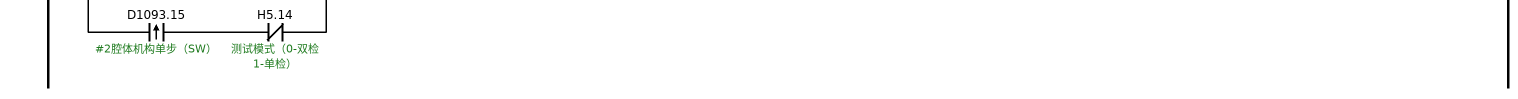
; [picture p240: 氦检机构 / 氦检腔2自动, rungs 7-7]
; rung 7: #2腔体机构步进条件（自动步）
LD D1096.00  ; #2腔体机构自动开始（自动步）
AND T1550  ; #2腔体机构开始运行条件延时(自动步)
LD D1096.01  ; #2腔体机构平移气缸到氦检位/数据初始化（自动步）
ANDNOT 802.01  ; #2腔体平移一级气缸缩回位标志[0002.01]
AND 802.02  ; #2腔体平移一级气缸伸出位标志[0002.02]
AND 802.03  ; #2腔体平移二级气缸缩回位标志[0002.03]
ANDNOT 802.04  ; #2腔体平移二级气缸伸出位标志[0002.04]
AND T1551  ; #2腔体机构数据初始化延时（自动步）
ORLD
LD D1096.02  ; #2腔体机构腔体顶升气缸上升（自动步）
AND 802.05  ; #2腔体顶伸气缸上升位标志[0002.05]
ANDNOT 802.06  ; #2腔体顶伸气缸下降位标志[0002.06]
ORLD
LD D1096.03  ; #2腔体机构等待氦检阀打开条件及腔体抽气阀打开条件/开腔体阀（自动步）
AND 821.10  ; #2-1腔体阀开到位标志
AND 821.12  ; #2-2腔体阀开到位标志
ANDNOT H27.00  ; #1腔体有清氦需求
ANDNOT H37.00  ; #3腔体有清氦需求
AND D1092.15  ; #2腔体机构腔体抽气阀打开允许
AND D1092.14  ; #2腔体氦检阀打开允许条件
LD W380.15  ; 氦检仪漏率低于设定值（稳态）
OR H5.02  ; 氦检仪屏蔽
ANDLD
AND=L(301) D1104 #0  ; #2腔体机构清氦步序号
ORLD
OR D1096.04  ; #2腔体机构（自动步）
LD D1096.05  ; #2腔体机构腔体抽气阀打开/延时开电池抽气阀（自动步）
LD T2000  ; #2-1腔体抽真空阈值到达延时（测试）
LD 823.08  ; #2-1电池抽真空阀开到位标志
AND T2020  ; #2-1电池抽真空阈值到达延时（测试）
LD H31.00  ; #2-1电池泄漏
ANDNOT H31.01  ; #2-2电池泄漏
ORLD
ORNOT H30.00  ; #2-1腔体有料记忆
LD 823.10  ; #2-2电池抽真空阀开到位标志
AND T2320  ; #2-2电池抽真空阈值到达延时（测试）
LDNOT H31.00  ; #2-1电池泄漏
AND H31.01  ; #2-2电池泄漏
ORLD
ORNOT H30.01  ; #2-2腔体有料记忆
ANDLD
OR H5.15  ; 腔体模式（0-正压 1-负压）
OR H5.10  ; 空跑程序
ANDLD
LD H31.04  ; #2-1腔体抽真空NG
ORNOT H30.00  ; #2-1腔体有料记忆
LD H31.05  ; #2-2腔体抽真空NG
ORNOT H30.01  ; #2-2腔体有料记忆
ANDLD
ORLD
LD H31.00  ; #2-1电池泄漏
AND H31.01  ; #2-2电池泄漏
ORLD
ANDLD
ORLD
LD D1096.06  ; #2腔体机构关电池抽气阀（自动步）  // 单个电池出现电池泄漏时，需将对应的腔体阀门关闭
ANDNOT W407.14  ; 设备氦气压力信号[alm]
ANDNOT W407.15  ; 精密调压阀信号[alm]
AND 823.09  ; #2-1电池抽真空阀关到位标志
AND 823.11  ; #2-2电池抽真空阀关到位标志
ANDNOT H31.04  ; #2-1腔体抽真空NG
ANDNOT H31.05  ; #2-2腔体抽真空NG
LD H31.00  ; #2-1电池泄漏
AND 821.11  ; #2-1腔体阀关到位标志
ORNOT H31.00  ; #2-1电池泄漏
ORNOT H30.00  ; #2-1腔体有料记忆
ANDLD
LD H31.01  ; #2-2电池泄漏
AND 821.13  ; #2-2腔体阀关到位标志
ORNOT H31.01  ; #2-2电池泄漏
ORNOT H30.01  ; #2-2腔体有料记忆
ANDLD
ORLD
LD D1096.07  ; #2腔体机构开电池注氦阀（自动步）  // 单个电池出现注氦超时时，需将对应的腔体阀门关闭
LD 823.12  ; #2-1电池注氦阀开到位标志
AND T2024  ; #2-1电池注氦压力到达延时（测试）
OR H31.00  ; #2-1电池泄漏
LD H31.02  ; #2-1电池注氦超时
AND 821.11  ; #2-1腔体阀关到位标志
ORLD
ORNOT H30.00  ; #2-1腔体有料记忆
LD 823.14  ; #2-2电池注氦阀开到位标志
AND T2324  ; #2-2电池注氦压力到达延时（测试）
OR H31.01  ; #2-2电池泄漏
LD H31.03  ; #2-2电池注氦超时
AND 821.13  ; #2-2腔体阀关到位标志
ORLD
ORNOT H30.01  ; #2-2腔体有料记忆
ANDLD
OR H5.15  ; 腔体模式（0-正压 1-负压）
OR H5.10  ; 空跑程序
ANDLD
ORLD
LD D1096.08  ; #2腔体机构关电池注氦阀（自动步）
AND 823.13  ; #2-1电池注氦阀关到位标志
AND 823.15  ; #2-2电池注氦阀关到位标志
LDNOT H31.03  ; #2-2电池注氦超时
ORNOT H31.02  ; #2-1电池注氦超时
ANDLD
ORLD
OR D1096.09  ; #2腔体机构（自动步）
LD D1096.10  ; #2腔体机构开腔体氦检阀/延时关腔体抽气阀（自动步）
LD T2006  ; #2-1腔体氦检数据取值判定延时（测试）
LD 820.10  ; 氦检仪真空阀开到位标志
AND 802.07  ; #2腔体氦检阀开到位标志[0002.07]
OR H5.02  ; 氦检仪屏蔽
ANDLD
LD H31.06  ; #2-1腔体氦检时腔体压力过高
AND H31.07  ; #2-2腔体氦检时腔体压力过高
ORLD
ANDLD
ORLD
OR D1096.11  ; #2腔体机构（自动步）
LD D1096.12  ; #2腔体机构关腔体氦检阀（自动步）
AND 802.08  ; #2腔体氦检阀关到位标志[0002.08]
ANDNOT 802.07  ; #2腔体氦检阀开到位标志[0002.07]
ORLD
OR D1096.13  ; #2腔体机构（自动步）
LD D1096.14  ; #2腔体机构开腔体#2-1腔体阀/开腔体#2-2腔体阀（自动步）
AND 821.10  ; #2-1腔体阀开到位标志
AND 821.12  ; #2-2腔体阀开到位标志
AND 802.08  ; #2腔体氦检阀关到位标志[0002.08]
ANDNOT H5.15  ; 腔体模式（0-正压 1-负压）
AND D1092.15  ; #2腔体机构腔体抽气阀打开允许
ORLD
LD D1096.15  ; #2腔体机构开腔体抽真空阀/开电池抽真空阀（自动步）
LD T2007  ; #2-1腔体抽残气压力到达延时（测试）
OR T2008  ; #2-1腔体抽残气时间上限到达延时（测试）
ANDLD
LD T2026  ; #2-1电池抽残气压力到达延时（测试）
OR T2027  ; #2-1电池抽残气时间上限到达延时（测试）
ORNOT H30.00  ; #2-1腔体有料记忆
LD T2326  ; #2-2电池抽残气压力到达延时（测试）
OR T2327  ; #2-2电池抽残气时间上限到达延时（测试）
ORNOT H30.01  ; #2-2腔体有料记忆
ANDLD
OR H5.10  ; 空跑程序
ANDLD
ORLD
LD D1097.00  ; #2腔体机构关腔体抽真空阀/关电池抽真空阀/开腔体阀（自动步）
AND 821.09  ; #2腔体抽真空阀关到位标志
AND 821.10  ; #2-1腔体阀开到位标志
AND 821.12  ; #2-2腔体阀开到位标志
AND 823.09  ; #2-1电池抽真空阀关到位标志
AND 823.11  ; #2-2电池抽真空阀关到位标志
ORLD
LD D1097.01  ; #2腔体机构清氦需求判定（自动步）
ANDNOT H32.00  ; #2腔体有清氦需求
ORLD
LD D1097.02  ; #2腔体机构开腔体破真空阀/开电池破真空阀（自动步）
AND T2002  ; #2-1腔体破真空阈值到达延时（测试）
LD T2022  ; #2-1电池破真空阈值到达延时（测试）
AND T2322  ; #2-2电池破真空阈值到达延时（测试）
OR H5.15  ; 腔体模式（0-正压 1-负压）
ANDLD
ORLD
LD D1097.03  ; #2腔体机构关腔体破真空阀/关电池破真空阀（自动步）
AND 821.15  ; #2腔体破真空阀关到位标志
AND 824.01  ; #2-1电池破真空阀关到位标志
AND 824.03  ; #2-2电池破真空阀关到位标志
ORLD
LD D1097.04  ; #2腔体机构复测需求判定（自动步）
ANDNOT H32.05  ; 腔体有复测需求
ORLD
OR D1097.05  ; #2腔体机构（自动步）
LD D1097.06  ; #2腔体机构腔体顶升气缸下降（自动步）
ANDNOT 802.05  ; #2腔体顶伸气缸上升位标志[0002.05]
AND 802.06  ; #2腔体顶伸气缸下降位标志[0002.06]
AND D1092.00  ; #2腔体机构平移气缸安全移动条件
LD H30.06  ; #2-1腔体测试完成记忆
ORNOT H30.00  ; #2-1腔体有料记忆
ANDLD
LD H30.07  ; #2-2腔体测试完成记忆
ORNOT H30.01  ; #2-2腔体有料记忆
ANDLD
ORLD
OR D1097.07  ; #2腔体机构（自动步）
LD D1097.08  ; #2腔体机构腔体平移气缸到出料位（自动步）
AND 802.01  ; #2腔体平移一级气缸缩回位标志[0002.01]
ANDNOT 802.02  ; #2腔体平移一级气缸伸出位标志[0002.02]
AND 802.03  ; #2腔体平移二级气缸缩回位标志[0002.03]
ANDNOT 802.04  ; #2腔体平移二级气缸伸出位标志[0002.04]
ORLD
LD D1097.09  ; #2腔体机构腔体等待取料完成信号（自动步）
ANDNOT H30.00  ; #2-1腔体有料记忆
ANDNOT H30.01  ; #2-2腔体有料记忆
AND D1092.00  ; #2腔体机构平移气缸安全移动条件
ORLD
OR D1097.10  ; #2腔体机构（自动步）
LD D1097.11  ; #2腔体机构平移气缸到上料位（自动步）
ANDNOT 802.01  ; #2腔体平移一级气缸缩回位标志[0002.01]
AND 802.02  ; #2腔体平移一级气缸伸出位标志[0002.02]
ANDNOT 802.03  ; #2腔体平移二级气缸缩回位标志[0002.03]
AND 802.04  ; #2腔体平移二级气缸伸出位标志[0002.04]
ORLD
OR D1097.12  ; #2腔体机构（自动步）
OR D1097.13  ; #2腔体机构（自动步）
OR D1097.14  ; #2腔体机构（自动步）
LD D1097.15  ; #2腔体机构循环结束（自动步）
AND P_Off
ORLD
LD D1094.01  ; #2腔体机构单步/自动循环运行中（自动步）
@LD D1093.15  ; #2腔体机构单步（SW）
ANDNOT H5.14  ; 测试模式（0-双检 1-单检）
ORLD
ANDLD
OUT D1095.01  ; #2腔体机构步进条件（自动步）

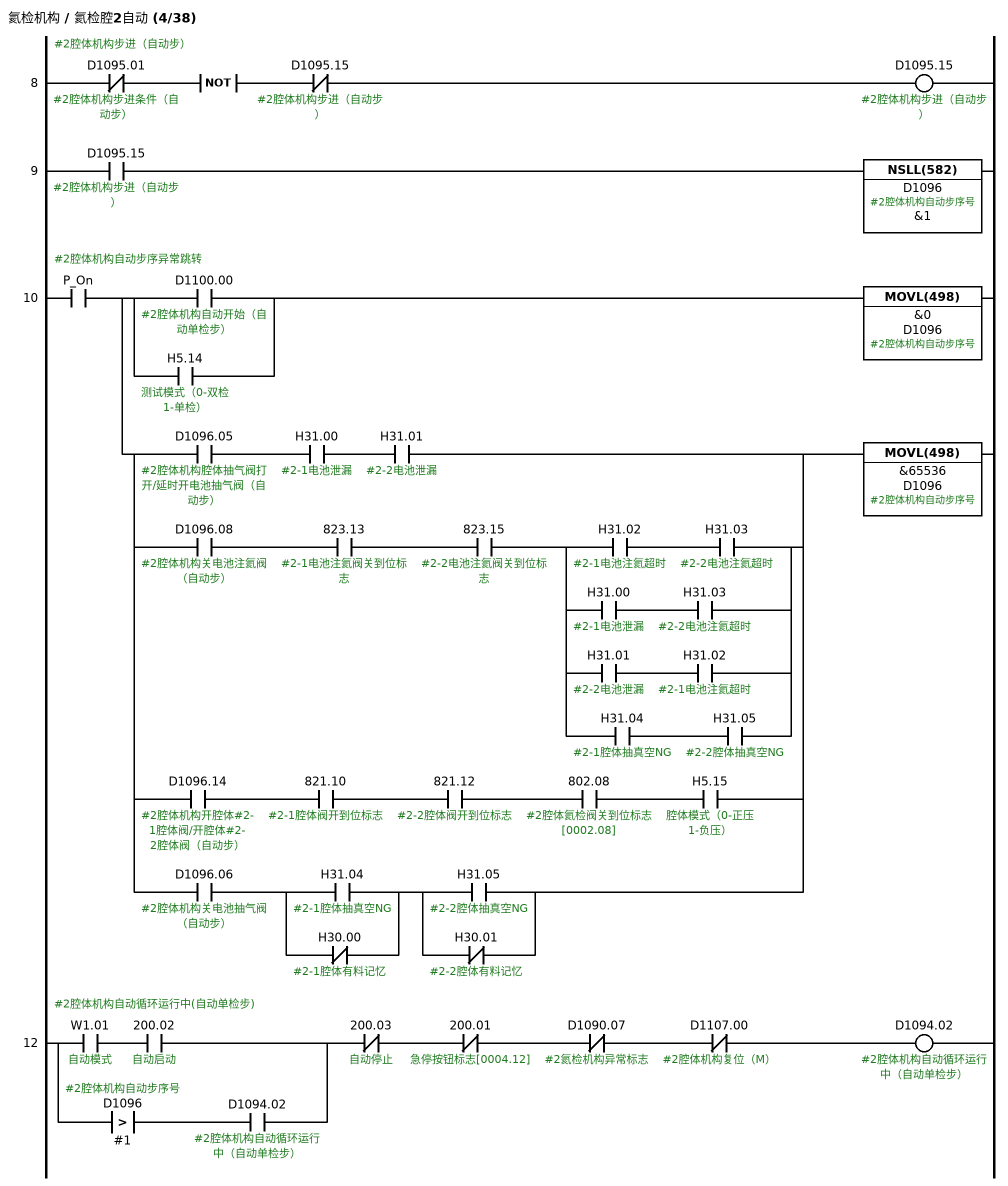
; rung 8: #2腔体机构步进（自动步）
LDNOT D1095.01  ; #2腔体机构步进条件（自动步）
NOT(520)
ANDNOT D1095.15  ; #2腔体机构步进（自动步）
OUT D1095.15  ; #2腔体机构步进（自动步）
; rung 9
LD D1095.15  ; #2腔体机构步进（自动步）
NSLL(582) D1096 &1  ; #2腔体机构自动步序号
; rung 10: #2腔体机构自动步序异常跳转
LD P_On
OUT TR0
LD D1100.00  ; #2腔体机构自动开始（自动单检步）
OR H5.14  ; 测试模式（0-双检 1-单检）
ANDLD
MOVL(498) &0 D1096  ; #2腔体机构自动步序号  // 测试模式为单检模式，腔体进入到复测步序时，将腔体机构自动步序清零
LD TR0
LD D1096.05  ; #2腔体机构腔体抽气阀打开/延时开电池抽气阀（自动步）
AND H31.00  ; #2-1电池泄漏
AND H31.01  ; #2-2电池泄漏
LD D1096.08  ; #2腔体机构关电池注氦阀（自动步）
AND 823.13  ; #2-1电池注氦阀关到位标志
AND 823.15  ; #2-2电池注氦阀关到位标志
LD H31.02  ; #2-1电池注氦超时
AND H31.03  ; #2-2电池注氦超时
LD H31.00  ; #2-1电池泄漏
AND H31.03  ; #2-2电池注氦超时
ORLD
LD H31.01  ; #2-2电池泄漏
AND H31.02  ; #2-1电池注氦超时
ORLD
LD H31.04  ; #2-1腔体抽真空NG
AND H31.05  ; #2-2腔体抽真空NG
ORLD
ANDLD
ORLD
LD D1096.14  ; #2腔体机构开腔体#2-1腔体阀/开腔体#2-2腔体阀（自动步）  // 负压模式不需要进行氦检后抽真空动作
AND 821.10  ; #2-1腔体阀开到位标志
AND 821.12  ; #2-2腔体阀开到位标志
AND 802.08  ; #2腔体氦检阀关到位标志[0002.08]
AND H5.15  ; 腔体模式（0-正压 1-负压）
ORLD
LD D1096.06  ; #2腔体机构关电池抽气阀（自动步）
LD H31.04  ; #2-1腔体抽真空NG
ORNOT H30.00  ; #2-1腔体有料记忆
ANDLD
LD H31.05  ; #2-2腔体抽真空NG
ORNOT H30.01  ; #2-2腔体有料记忆
ANDLD
ORLD
ANDLD
MOVL(498) &65536 D1096  ; #2腔体机构自动步序号  // 出现腔体抽真空NG，双电池抽真空NG，双电池注氦超时的情况，均跳转至自动步序D1067.0
; rung 11: ******************************* / 自动单检步序 / *******************************
; rung 12: #2腔体机构自动循环运行中(自动单检步)
LD W1.01  ; 自动模式
AND 200.02  ; 自动启动
LD>L(321) D1096 #1  ; #2腔体机构自动步序号
AND D1094.02  ; #2腔体机构自动循环运行中（自动单检步）
ORLD
ANDNOT 200.03  ; 自动停止
ANDNOT 200.01  ; 急停按钮标志[0004.12]
ANDNOT D1090.07  ; #2氦检机构异常标志
ANDNOT D1107.00  ; #2腔体机构复位（M）
OUT D1094.02  ; #2腔体机构自动循环运行中（自动单检步）

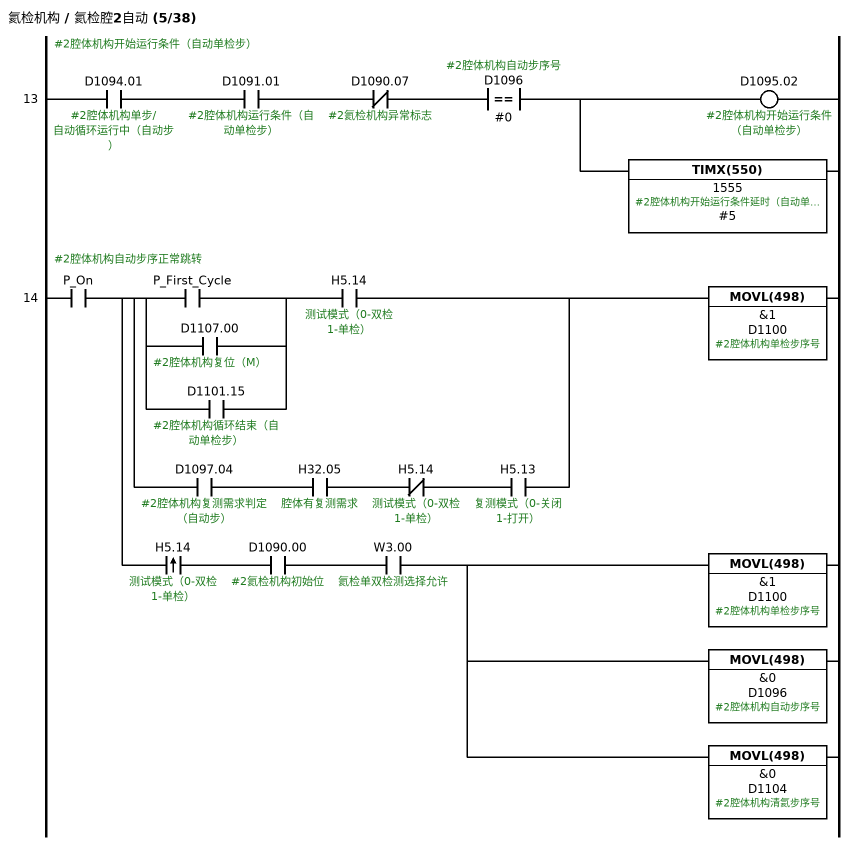
; rung 13: #2腔体机构开始运行条件（自动单检步）
LD D1094.01  ; #2腔体机构单步/自动循环运行中（自动步）
AND D1091.01  ; #2腔体机构运行条件（自动单检步）
ANDNOT D1090.07  ; #2氦检机构异常标志
AND=L(301) D1096 #0  ; #2腔体机构自动步序号
OUT D1095.02  ; #2腔体机构开始运行条件（自动单检步）
TIMX(550) 1555 #5  ; #2腔体机构开始运行条件延时（自动单检步）
; rung 14: #2腔体机构自动步序正常跳转
LD P_On
OUT TR0
LD P_First_Cycle
OR D1107.00  ; #2腔体机构复位（M）
OR D1101.15  ; #2腔体机构循环结束（自动单检步）
AND H5.14  ; 测试模式（0-双检 1-单检）
LD D1097.04  ; #2腔体机构复测需求判定（自动步）
AND H32.05  ; 腔体有复测需求
ANDNOT H5.14  ; 测试模式（0-双检 1-单检）
AND H5.13  ; 复测模式（0-关闭 1-打开）
ORLD
ANDLD
MOVL(498) &1 D1100  ; #2腔体机构单检步序号
LD TR0
@AND H5.14  ; 测试模式（0-双检 1-单检）
AND D1090.00  ; #2氦检机构初始位
AND W3.00  ; 氦检单双检测选择允许
MOVL(498) &1 D1100  ; #2腔体机构单检步序号
MOVL(498) &0 D1096  ; #2腔体机构自动步序号
MOVL(498) &0 D1104  ; #2腔体机构清氦步序号

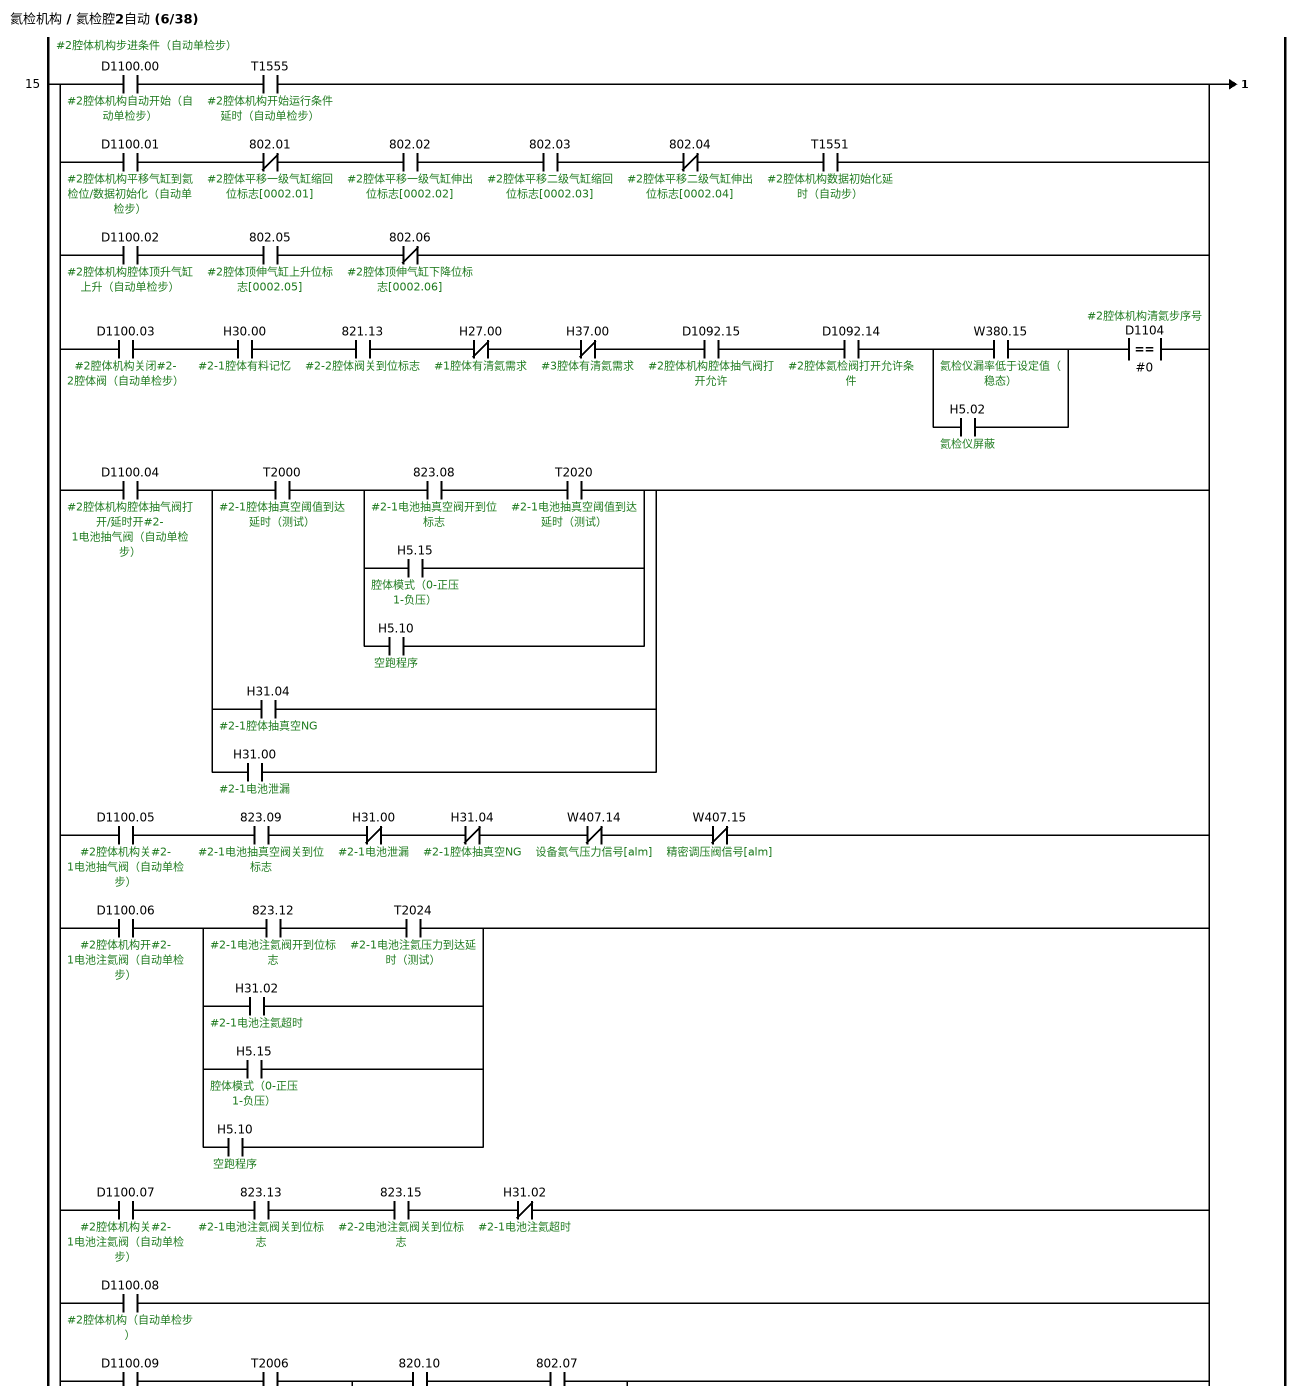

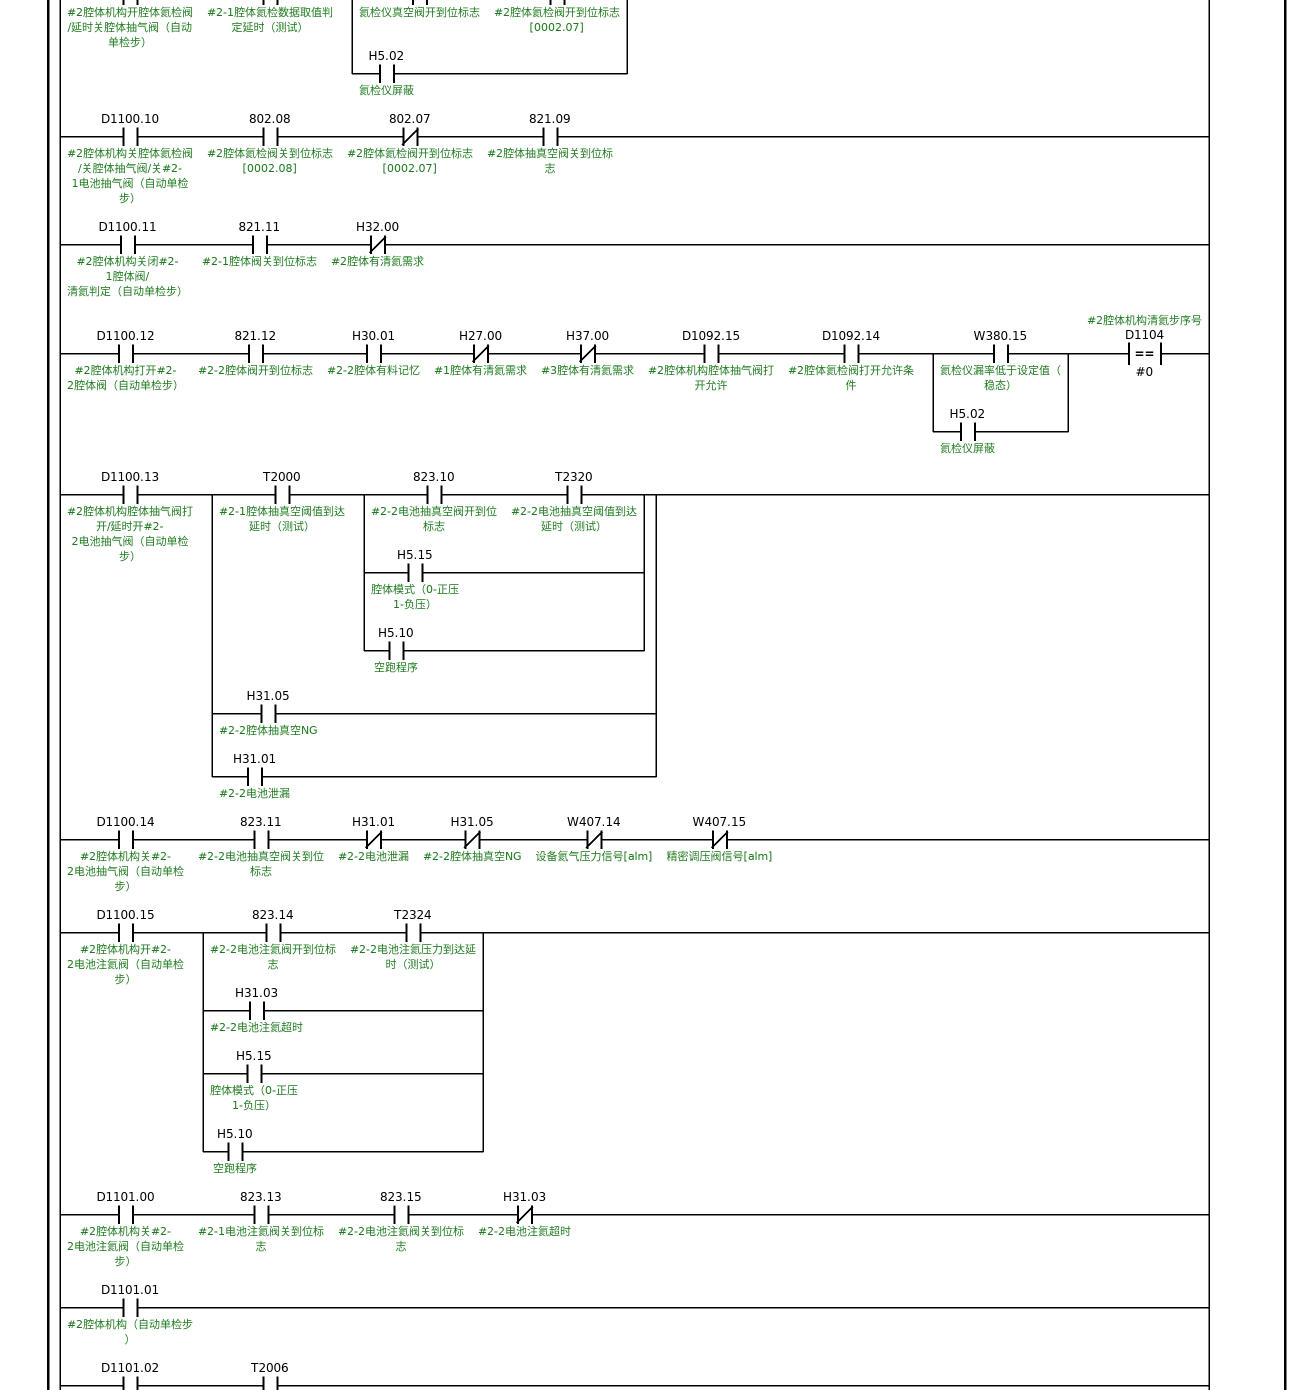

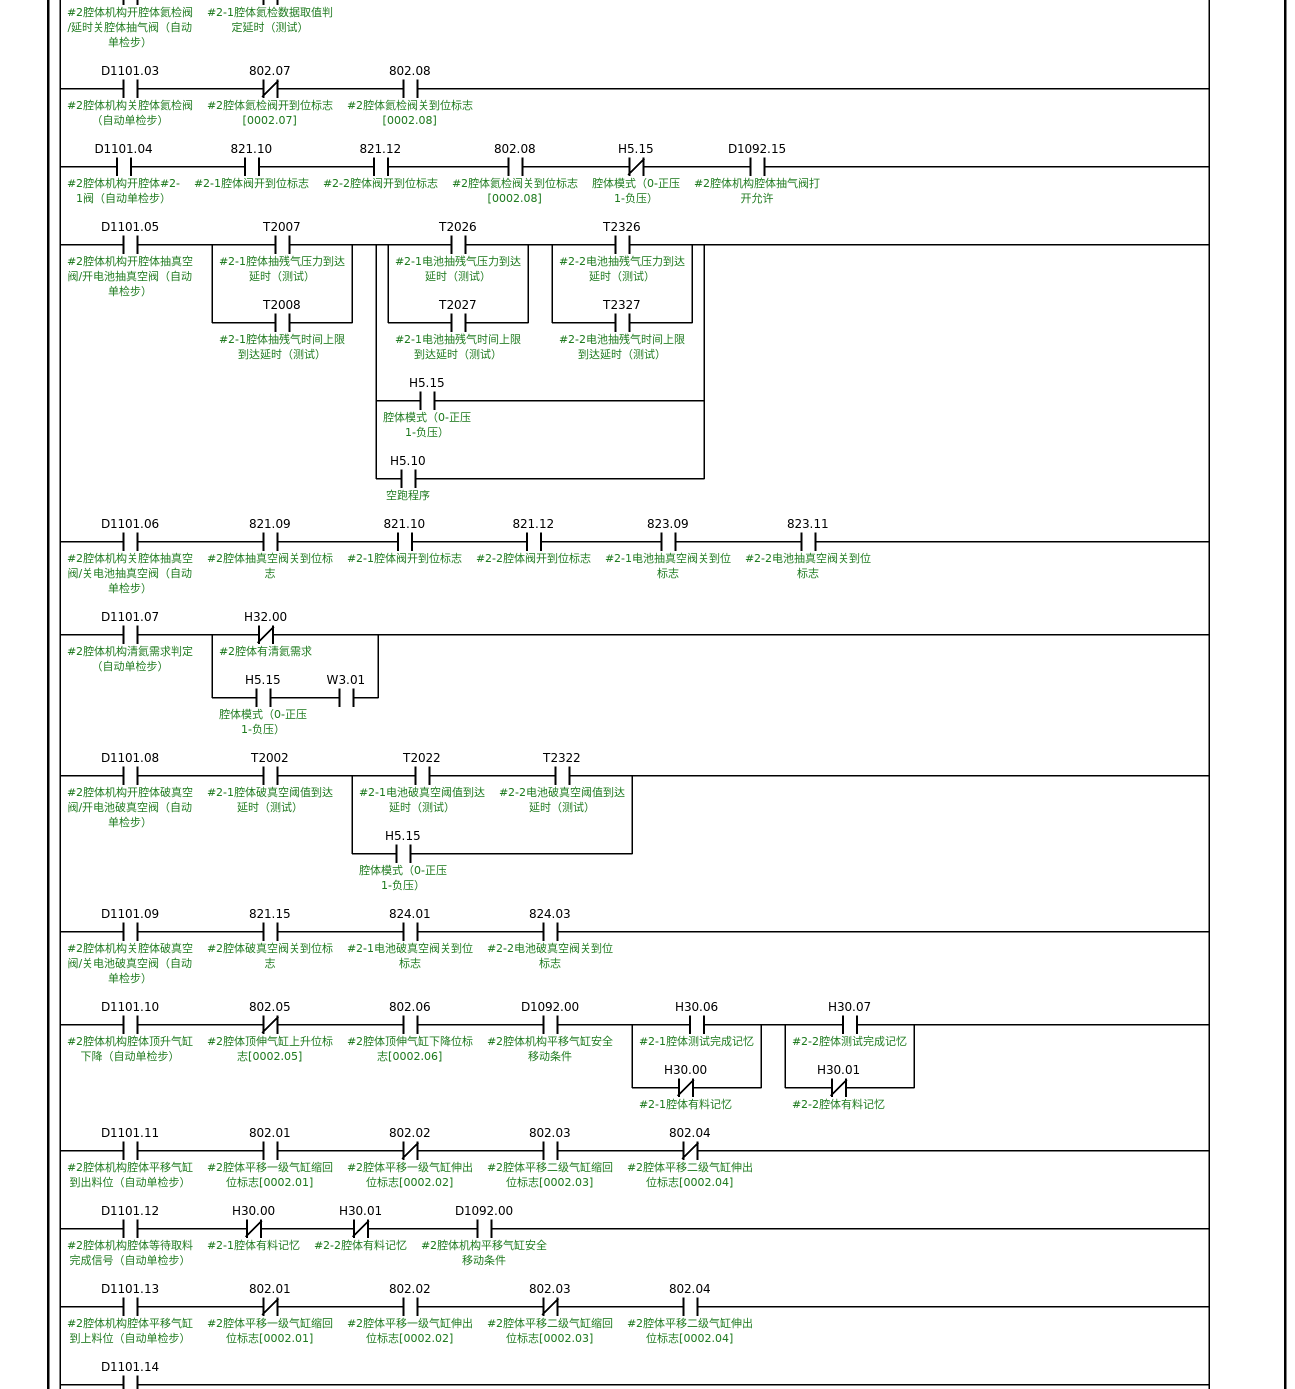

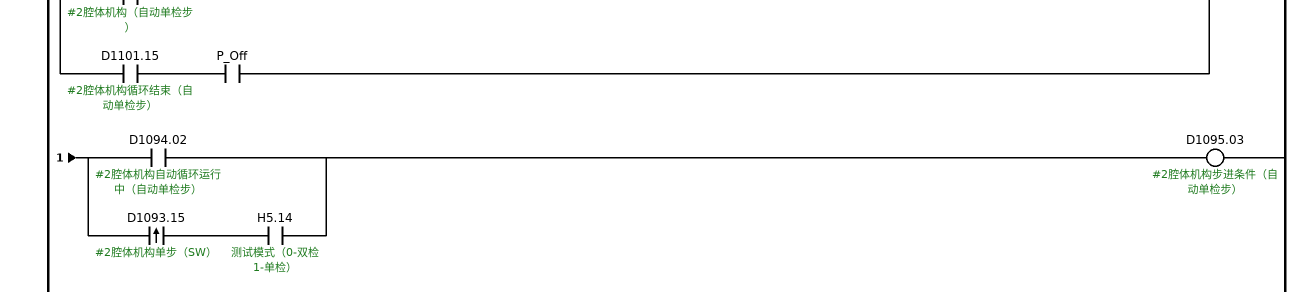
; rung 15: #2腔体机构步进条件（自动单检步）
LD D1100.00  ; #2腔体机构自动开始（自动单检步）
AND T1555  ; #2腔体机构开始运行条件延时（自动单检步）
LD D1100.01  ; #2腔体机构平移气缸到氦检位/数据初始化（自动单检步）
ANDNOT 802.01  ; #2腔体平移一级气缸缩回位标志[0002.01]
AND 802.02  ; #2腔体平移一级气缸伸出位标志[0002.02]
AND 802.03  ; #2腔体平移二级气缸缩回位标志[0002.03]
ANDNOT 802.04  ; #2腔体平移二级气缸伸出位标志[0002.04]
AND T1551  ; #2腔体机构数据初始化延时（自动步）
ORLD
LD D1100.02  ; #2腔体机构腔体顶升气缸上升（自动单检步）
AND 802.05  ; #2腔体顶伸气缸上升位标志[0002.05]
ANDNOT 802.06  ; #2腔体顶伸气缸下降位标志[0002.06]
ORLD
LD D1100.03  ; #2腔体机构关闭#2-2腔体阀（自动单检步）
AND H30.00  ; #2-1腔体有料记忆
AND 821.13  ; #2-2腔体阀关到位标志
ANDNOT H27.00  ; #1腔体有清氦需求
ANDNOT H37.00  ; #3腔体有清氦需求
AND D1092.15  ; #2腔体机构腔体抽气阀打开允许
AND D1092.14  ; #2腔体氦检阀打开允许条件
LD W380.15  ; 氦检仪漏率低于设定值（稳态）
OR H5.02  ; 氦检仪屏蔽
ANDLD
AND=L(301) D1104 #0  ; #2腔体机构清氦步序号
ORLD
LD D1100.04  ; #2腔体机构腔体抽气阀打开/延时开#2-1电池抽气阀（自动单检步）
LD T2000  ; #2-1腔体抽真空阈值到达延时（测试）
LD 823.08  ; #2-1电池抽真空阀开到位标志
AND T2020  ; #2-1电池抽真空阈值到达延时（测试）
OR H5.15  ; 腔体模式（0-正压 1-负压）
OR H5.10  ; 空跑程序
ANDLD
OR H31.04  ; #2-1腔体抽真空NG
OR H31.00  ; #2-1电池泄漏
ANDLD
ORLD
LD D1100.05  ; #2腔体机构关#2-1电池抽气阀（自动单检步）
AND 823.09  ; #2-1电池抽真空阀关到位标志
ANDNOT H31.00  ; #2-1电池泄漏
ANDNOT H31.04  ; #2-1腔体抽真空NG
ANDNOT W407.14  ; 设备氦气压力信号[alm]
ANDNOT W407.15  ; 精密调压阀信号[alm]
ORLD
LD D1100.06  ; #2腔体机构开#2-1电池注氦阀（自动单检步）
LD 823.12  ; #2-1电池注氦阀开到位标志
AND T2024  ; #2-1电池注氦压力到达延时（测试）
OR H31.02  ; #2-1电池注氦超时
OR H5.15  ; 腔体模式（0-正压 1-负压）
OR H5.10  ; 空跑程序
ANDLD
ORLD
LD D1100.07  ; #2腔体机构关#2-1电池注氦阀（自动单检步）
AND 823.13  ; #2-1电池注氦阀关到位标志
AND 823.15  ; #2-2电池注氦阀关到位标志
ANDNOT H31.02  ; #2-1电池注氦超时
ORLD
OR D1100.08  ; #2腔体机构（自动单检步）
LD D1100.09  ; #2腔体机构开腔体氦检阀/延时关腔体抽气阀（自动单检步）
AND T2006  ; #2-1腔体氦检数据取值判定延时（测试）
LD 820.10  ; 氦检仪真空阀开到位标志
AND 802.07  ; #2腔体氦检阀开到位标志[0002.07]
OR H5.02  ; 氦检仪屏蔽
ANDLD
ORLD
LD D1100.10  ; #2腔体机构关腔体氦检阀/关腔体抽气阀/关#2-1电池抽气阀（自动单检步）
AND 802.08  ; #2腔体氦检阀关到位标志[0002.08]
ANDNOT 802.07  ; #2腔体氦检阀开到位标志[0002.07]
AND 821.09  ; #2腔体抽真空阀关到位标志
ORLD
LD D1100.11  ; #2腔体机构关闭#2-1腔体阀/清氦判定（自动单检步）
AND 821.11  ; #2-1腔体阀关到位标志
ANDNOT H32.00  ; #2腔体有清氦需求
ORLD
LD D1100.12  ; #2腔体机构打开#2-2腔体阀（自动单检步）
AND 821.12  ; #2-2腔体阀开到位标志
AND H30.01  ; #2-2腔体有料记忆
ANDNOT H27.00  ; #1腔体有清氦需求
ANDNOT H37.00  ; #3腔体有清氦需求
AND D1092.15  ; #2腔体机构腔体抽气阀打开允许
AND D1092.14  ; #2腔体氦检阀打开允许条件
LD W380.15  ; 氦检仪漏率低于设定值（稳态）
OR H5.02  ; 氦检仪屏蔽
ANDLD
AND=L(301) D1104 #0  ; #2腔体机构清氦步序号
ORLD
LD D1100.13  ; #2腔体机构腔体抽气阀打开/延时开#2-2电池抽气阀（自动单检步）
LD T2000  ; #2-1腔体抽真空阈值到达延时（测试）
LD 823.10  ; #2-2电池抽真空阀开到位标志
AND T2320  ; #2-2电池抽真空阈值到达延时（测试）
OR H5.15  ; 腔体模式（0-正压 1-负压）
OR H5.10  ; 空跑程序
ANDLD
OR H31.05  ; #2-2腔体抽真空NG
OR H31.01  ; #2-2电池泄漏
ANDLD
ORLD
LD D1100.14  ; #2腔体机构关#2-2电池抽气阀（自动单检步）
AND 823.11  ; #2-2电池抽真空阀关到位标志
ANDNOT H31.01  ; #2-2电池泄漏
ANDNOT H31.05  ; #2-2腔体抽真空NG
ANDNOT W407.14  ; 设备氦气压力信号[alm]
ANDNOT W407.15  ; 精密调压阀信号[alm]
ORLD
LD D1100.15  ; #2腔体机构开#2-2电池注氦阀（自动单检步）
LD 823.14  ; #2-2电池注氦阀开到位标志
AND T2324  ; #2-2电池注氦压力到达延时（测试）
OR H31.03  ; #2-2电池注氦超时
OR H5.15  ; 腔体模式（0-正压 1-负压）
OR H5.10  ; 空跑程序
ANDLD
ORLD
LD D1101.00  ; #2腔体机构关#2-2电池注氦阀（自动单检步）
AND 823.13  ; #2-1电池注氦阀关到位标志
AND 823.15  ; #2-2电池注氦阀关到位标志
ANDNOT H31.03  ; #2-2电池注氦超时
ORLD
OR D1101.01  ; #2腔体机构（自动单检步）
LD D1101.02  ; #2腔体机构开腔体氦检阀/延时关腔体抽气阀（自动单检步）
AND T2006  ; #2-1腔体氦检数据取值判定延时（测试）
ORLD
LD D1101.03  ; #2腔体机构关腔体氦检阀（自动单检步）
ANDNOT 802.07  ; #2腔体氦检阀开到位标志[0002.07]
AND 802.08  ; #2腔体氦检阀关到位标志[0002.08]
ORLD
LD D1101.04  ; #2腔体机构开腔体#2-1阀（自动单检步）
AND 821.10  ; #2-1腔体阀开到位标志
AND 821.12  ; #2-2腔体阀开到位标志
AND 802.08  ; #2腔体氦检阀关到位标志[0002.08]
ANDNOT H5.15  ; 腔体模式（0-正压 1-负压）
AND D1092.15  ; #2腔体机构腔体抽气阀打开允许
ORLD
LD D1101.05  ; #2腔体机构开腔体抽真空阀/开电池抽真空阀（自动单检步）
LD T2007  ; #2-1腔体抽残气压力到达延时（测试）
OR T2008  ; #2-1腔体抽残气时间上限到达延时（测试）
ANDLD
LD T2026  ; #2-1电池抽残气压力到达延时（测试）
OR T2027  ; #2-1电池抽残气时间上限到达延时（测试）
LD T2326  ; #2-2电池抽残气压力到达延时（测试）
OR T2327  ; #2-2电池抽残气时间上限到达延时（测试）
ANDLD
OR H5.15  ; 腔体模式（0-正压 1-负压）
OR H5.10  ; 空跑程序
ANDLD
ORLD
LD D1101.06  ; #2腔体机构关腔体抽真空阀/关电池抽真空阀（自动单检步）
AND 821.09  ; #2腔体抽真空阀关到位标志
AND 821.10  ; #2-1腔体阀开到位标志
AND 821.12  ; #2-2腔体阀开到位标志
AND 823.09  ; #2-1电池抽真空阀关到位标志
AND 823.11  ; #2-2电池抽真空阀关到位标志
ORLD
LD D1101.07  ; #2腔体机构清氦需求判定（自动单检步）
LDNOT H32.00  ; #2腔体有清氦需求
LD H5.15  ; 腔体模式（0-正压 1-负压）
AND W3.01
ORLD
ANDLD
ORLD
LD D1101.08  ; #2腔体机构开腔体破真空阀/开电池破真空阀（自动单检步）
AND T2002  ; #2-1腔体破真空阈值到达延时（测试）
LD T2022  ; #2-1电池破真空阈值到达延时（测试）
AND T2322  ; #2-2电池破真空阈值到达延时（测试）
OR H5.15  ; 腔体模式（0-正压 1-负压）
ANDLD
ORLD
LD D1101.09  ; #2腔体机构关腔体破真空阀/关电池破真空阀（自动单检步）
AND 821.15  ; #2腔体破真空阀关到位标志
AND 824.01  ; #2-1电池破真空阀关到位标志
AND 824.03  ; #2-2电池破真空阀关到位标志
ORLD
LD D1101.10  ; #2腔体机构腔体顶升气缸下降（自动单检步）
ANDNOT 802.05  ; #2腔体顶伸气缸上升位标志[0002.05]
AND 802.06  ; #2腔体顶伸气缸下降位标志[0002.06]
AND D1092.00  ; #2腔体机构平移气缸安全移动条件
LD H30.06  ; #2-1腔体测试完成记忆
ORNOT H30.00  ; #2-1腔体有料记忆
ANDLD
LD H30.07  ; #2-2腔体测试完成记忆
ORNOT H30.01  ; #2-2腔体有料记忆
ANDLD
ORLD
LD D1101.11  ; #2腔体机构腔体平移气缸到出料位（自动单检步）
AND 802.01  ; #2腔体平移一级气缸缩回位标志[0002.01]
ANDNOT 802.02  ; #2腔体平移一级气缸伸出位标志[0002.02]
AND 802.03  ; #2腔体平移二级气缸缩回位标志[0002.03]
ANDNOT 802.04  ; #2腔体平移二级气缸伸出位标志[0002.04]
ORLD
LD D1101.12  ; #2腔体机构腔体等待取料完成信号（自动单检步）
ANDNOT H30.00  ; #2-1腔体有料记忆
ANDNOT H30.01  ; #2-2腔体有料记忆
AND D1092.00  ; #2腔体机构平移气缸安全移动条件
ORLD
LD D1101.13  ; #2腔体机构腔体平移气缸到上料位（自动单检步）
ANDNOT 802.01  ; #2腔体平移一级气缸缩回位标志[0002.01]
AND 802.02  ; #2腔体平移一级气缸伸出位标志[0002.02]
ANDNOT 802.03  ; #2腔体平移二级气缸缩回位标志[0002.03]
AND 802.04  ; #2腔体平移二级气缸伸出位标志[0002.04]
ORLD
OR D1101.14  ; #2腔体机构（自动单检步）
LD D1101.15  ; #2腔体机构循环结束（自动单检步）
AND P_Off
ORLD
LD D1094.02  ; #2腔体机构自动循环运行中（自动单检步）
@LD D1093.15  ; #2腔体机构单步（SW）
AND H5.14  ; 测试模式（0-双检 1-单检）
ORLD
ANDLD
OUT D1095.03  ; #2腔体机构步进条件（自动单检步）

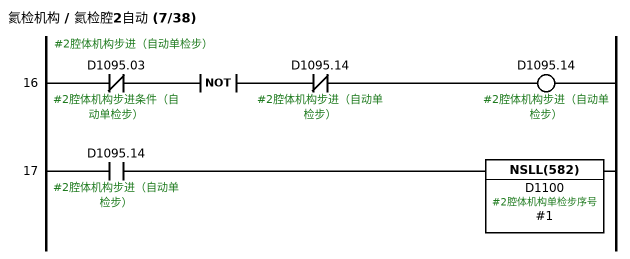
; rung 16: #2腔体机构步进（自动单检步）
LDNOT D1095.03  ; #2腔体机构步进条件（自动单检步）
NOT(520)
ANDNOT D1095.14  ; #2腔体机构步进（自动单检步）
OUT D1095.14  ; #2腔体机构步进（自动单检步）
; rung 17
LD D1095.14  ; #2腔体机构步进（自动单检步）
NSLL(582) D1100 #1  ; #2腔体机构单检步序号

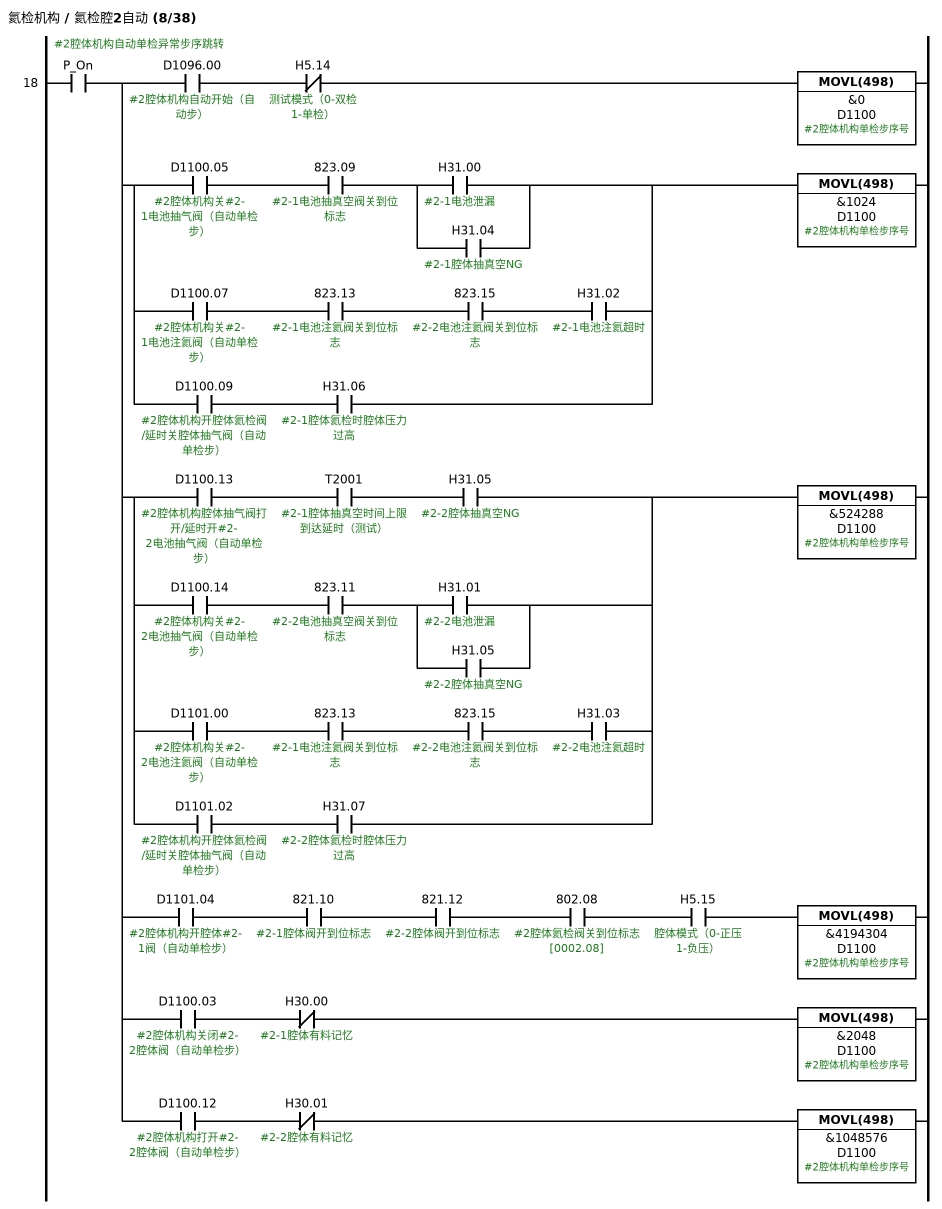
; rung 18: #2腔体机构自动单检异常步序跳转
LD P_On
OUT TR0
AND D1096.00  ; #2腔体机构自动开始（自动步）
ANDNOT H5.14  ; 测试模式（0-双检 1-单检）
MOVL(498) &0 D1100  ; #2腔体机构单检步序号
LD TR0
LD D1100.05  ; #2腔体机构关#2-1电池抽气阀（自动单检步）
AND 823.09  ; #2-1电池抽真空阀关到位标志
LD H31.00  ; #2-1电池泄漏
OR H31.04  ; #2-1腔体抽真空NG
ANDLD
LD D1100.07  ; #2腔体机构关#2-1电池注氦阀（自动单检步）
AND 823.13  ; #2-1电池注氦阀关到位标志
AND 823.15  ; #2-2电池注氦阀关到位标志
AND H31.02  ; #2-1电池注氦超时
ORLD
LD D1100.09  ; #2腔体机构开腔体氦检阀/延时关腔体抽气阀（自动单检步）  // 氦检阀开启后腔体压力超过安全阀值，测试判定为NG（氦检异常）
AND H31.06  ; #2-1腔体氦检时腔体压力过高
ORLD
ANDLD
MOVL(498) &1024 D1100  ; #2腔体机构单检步序号  // #1-1腔体出现腔体泄漏，电池泄漏，注氦超时的情况，均跳转至单检步序D1070.10
LD TR0
LD D1100.13  ; #2腔体机构腔体抽气阀打开/延时开#2-2电池抽气阀（自动单检步）
AND T2001  ; #2-1腔体抽真空时间上限到达延时（测试）
AND H31.05  ; #2-2腔体抽真空NG
LD D1100.14  ; #2腔体机构关#2-2电池抽气阀（自动单检步）
AND 823.11  ; #2-2电池抽真空阀关到位标志
LD H31.01  ; #2-2电池泄漏
OR H31.05  ; #2-2腔体抽真空NG
ANDLD
ORLD
LD D1101.00  ; #2腔体机构关#2-2电池注氦阀（自动单检步）
AND 823.13  ; #2-1电池注氦阀关到位标志
AND 823.15  ; #2-2电池注氦阀关到位标志
AND H31.03  ; #2-2电池注氦超时
ORLD
LD D1101.02  ; #2腔体机构开腔体氦检阀/延时关腔体抽气阀（自动单检步）  // 氦检阀开启后腔体压力超过安全阀值，测试判定为NG（氦检异常）
AND H31.07  ; #2-2腔体氦检时腔体压力过高
ORLD
ANDLD
MOVL(498) &524288 D1100  ; #2腔体机构单检步序号  // #1-2腔体出现腔体泄漏，电池泄漏，注氦超时的情况，均跳转至单检步序D1071.03
LD TR0
AND D1101.04  ; #2腔体机构开腔体#2-1阀（自动单检步）
AND 821.10  ; #2-1腔体阀开到位标志
AND 821.12  ; #2-2腔体阀开到位标志
AND 802.08  ; #2腔体氦检阀关到位标志[0002.08]
AND H5.15  ; 腔体模式（0-正压 1-负压）
MOVL(498) &4194304 D1100  ; #2腔体机构单检步序号  // 负压模式下步序正常流程步序不需要抽残气，直接跳转至D1071.06
LD TR0
AND D1100.03  ; #2腔体机构关闭#2-2腔体阀（自动单检步）
ANDNOT H30.00  ; #2-1腔体有料记忆
MOVL(498) &2048 D1100  ; #2腔体机构单检步序号  // 清尾料是#1-1无料，跳转至D1070.11
LD TR0
AND D1100.12  ; #2腔体机构打开#2-2腔体阀（自动单检步）
ANDNOT H30.01  ; #2-2腔体有料记忆
MOVL(498) &1048576 D1100  ; #2腔体机构单检步序号  // 清尾料时#1-2无料，跳转至D1071.04
; rung 19: ******************************* / 清氦步序 / *******************************

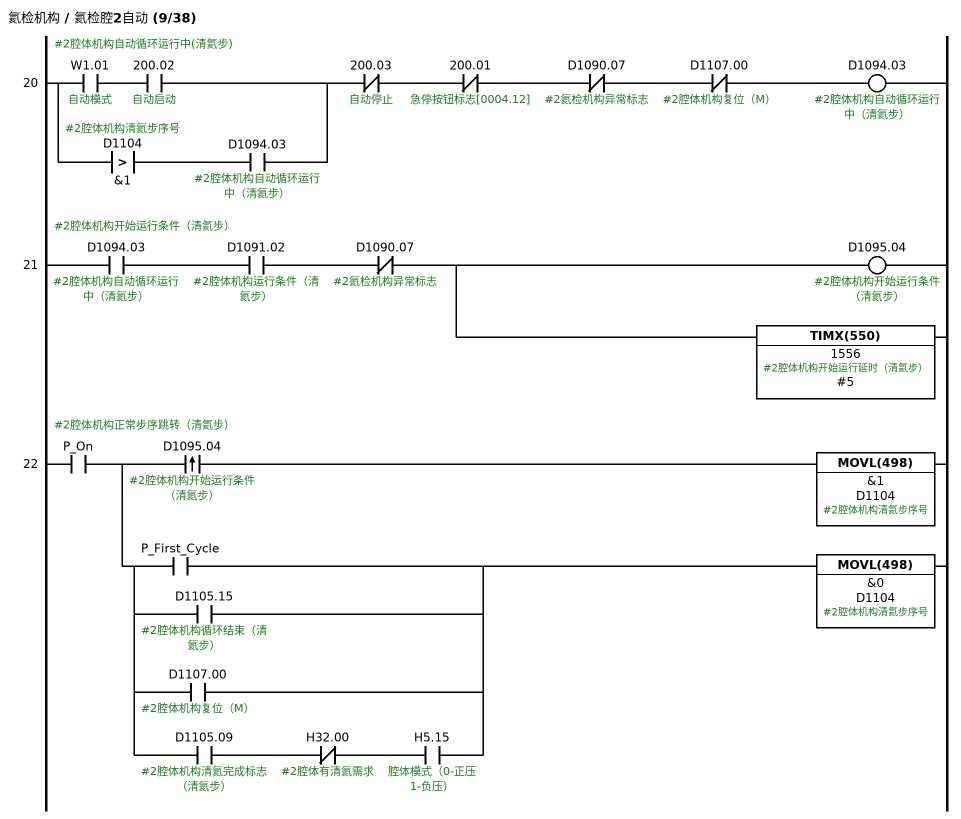
; rung 20: #2腔体机构自动循环运行中(清氦步)
LD W1.01  ; 自动模式
AND 200.02  ; 自动启动
LD>L(321) D1104 &1  ; #2腔体机构清氦步序号
AND D1094.03  ; #2腔体机构自动循环运行中（清氦步）
ORLD
ANDNOT 200.03  ; 自动停止
ANDNOT 200.01  ; 急停按钮标志[0004.12]
ANDNOT D1090.07  ; #2氦检机构异常标志
ANDNOT D1107.00  ; #2腔体机构复位（M）
OUT D1094.03  ; #2腔体机构自动循环运行中（清氦步）
; rung 21: #2腔体机构开始运行条件（清氦步）
LD D1094.03  ; #2腔体机构自动循环运行中（清氦步）
AND D1091.02  ; #2腔体机构运行条件（清氦步）
ANDNOT D1090.07  ; #2氦检机构异常标志
OUT D1095.04  ; #2腔体机构开始运行条件（清氦步）
TIMX(550) 1556 #5  ; #2腔体机构开始运行延时（清氦步）
; rung 22: #2腔体机构正常步序跳转（清氦步）
LD P_On
OUT TR0
@AND D1095.04  ; #2腔体机构开始运行条件（清氦步）
MOVL(498) &1 D1104  ; #2腔体机构清氦步序号
LD TR0
LD P_First_Cycle
OR D1105.15  ; #2腔体机构循环结束（清氦步）
OR D1107.00  ; #2腔体机构复位（M）
LD D1105.09  ; #2腔体机构清氦完成标志（清氦步）  // 正压腔体是待料清氦，需跳转回测试步序
ANDNOT H32.00  ; #2腔体有清氦需求
AND H5.15  ; 腔体模式（0-正压 1-负压）
ORLD
ANDLD
MOVL(498) &0 D1104  ; #2腔体机构清氦步序号

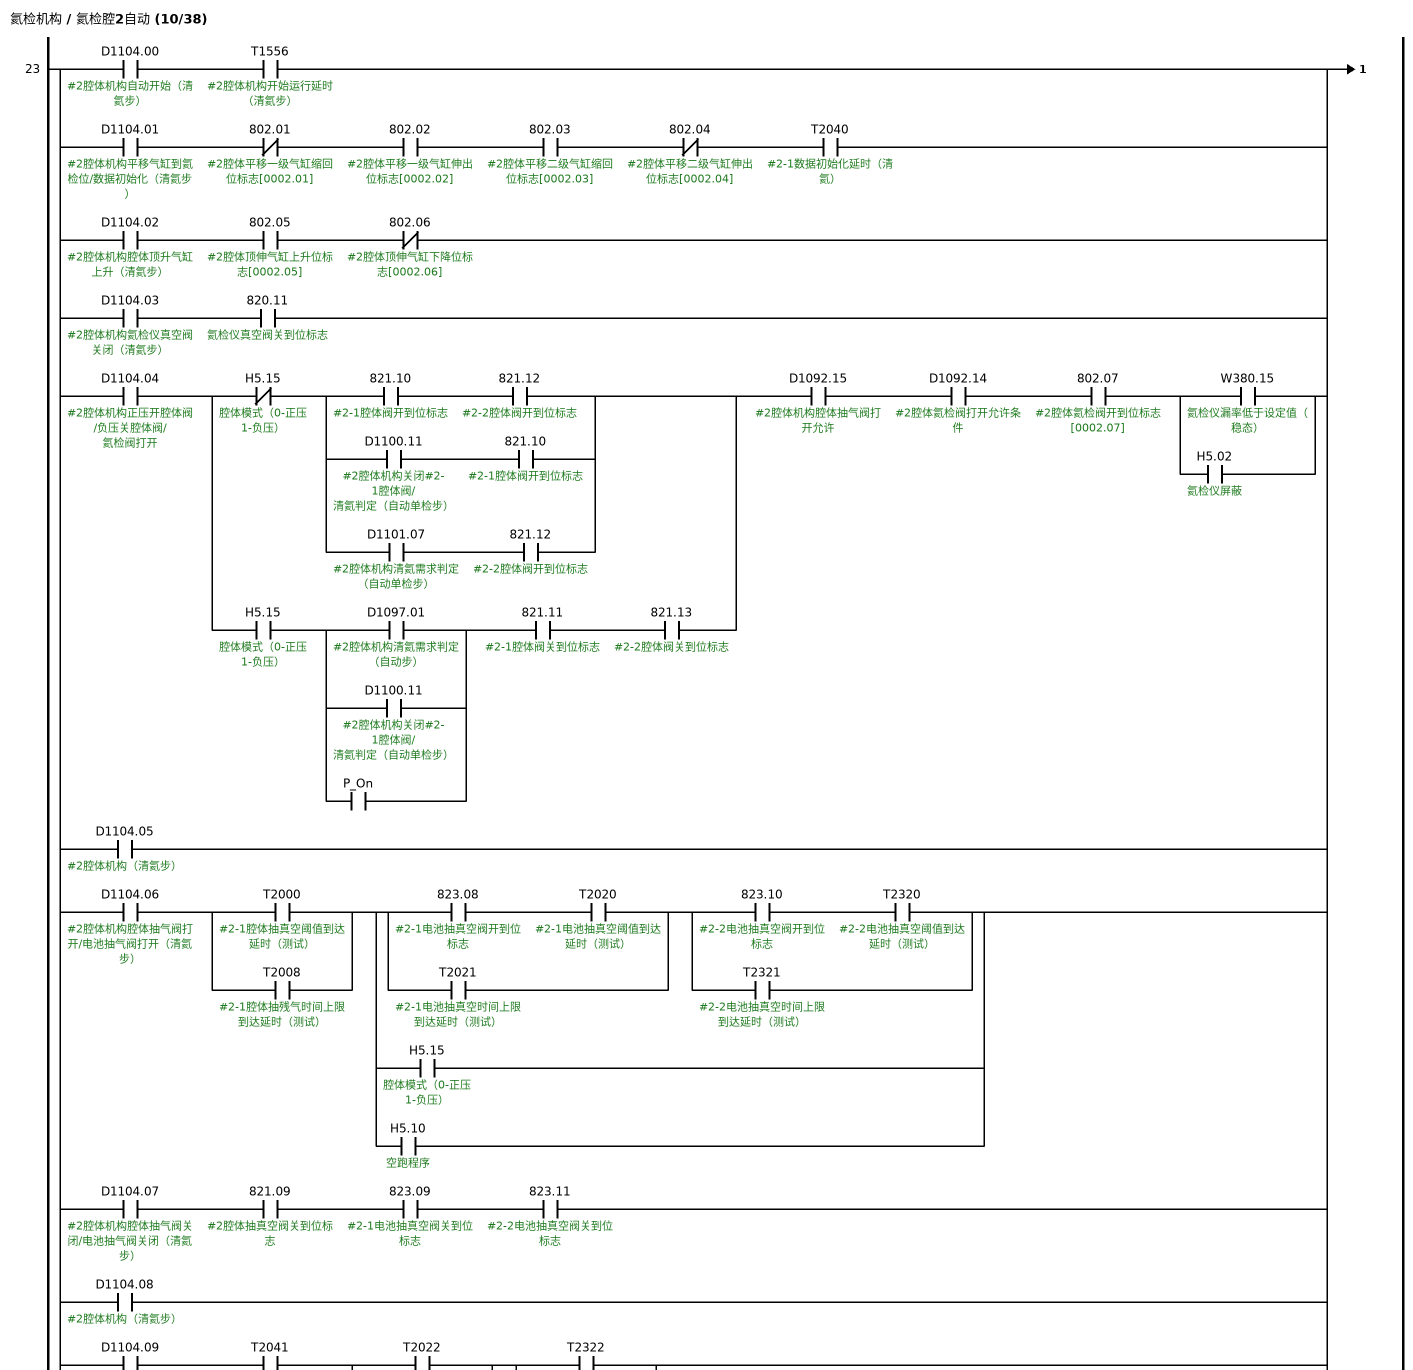

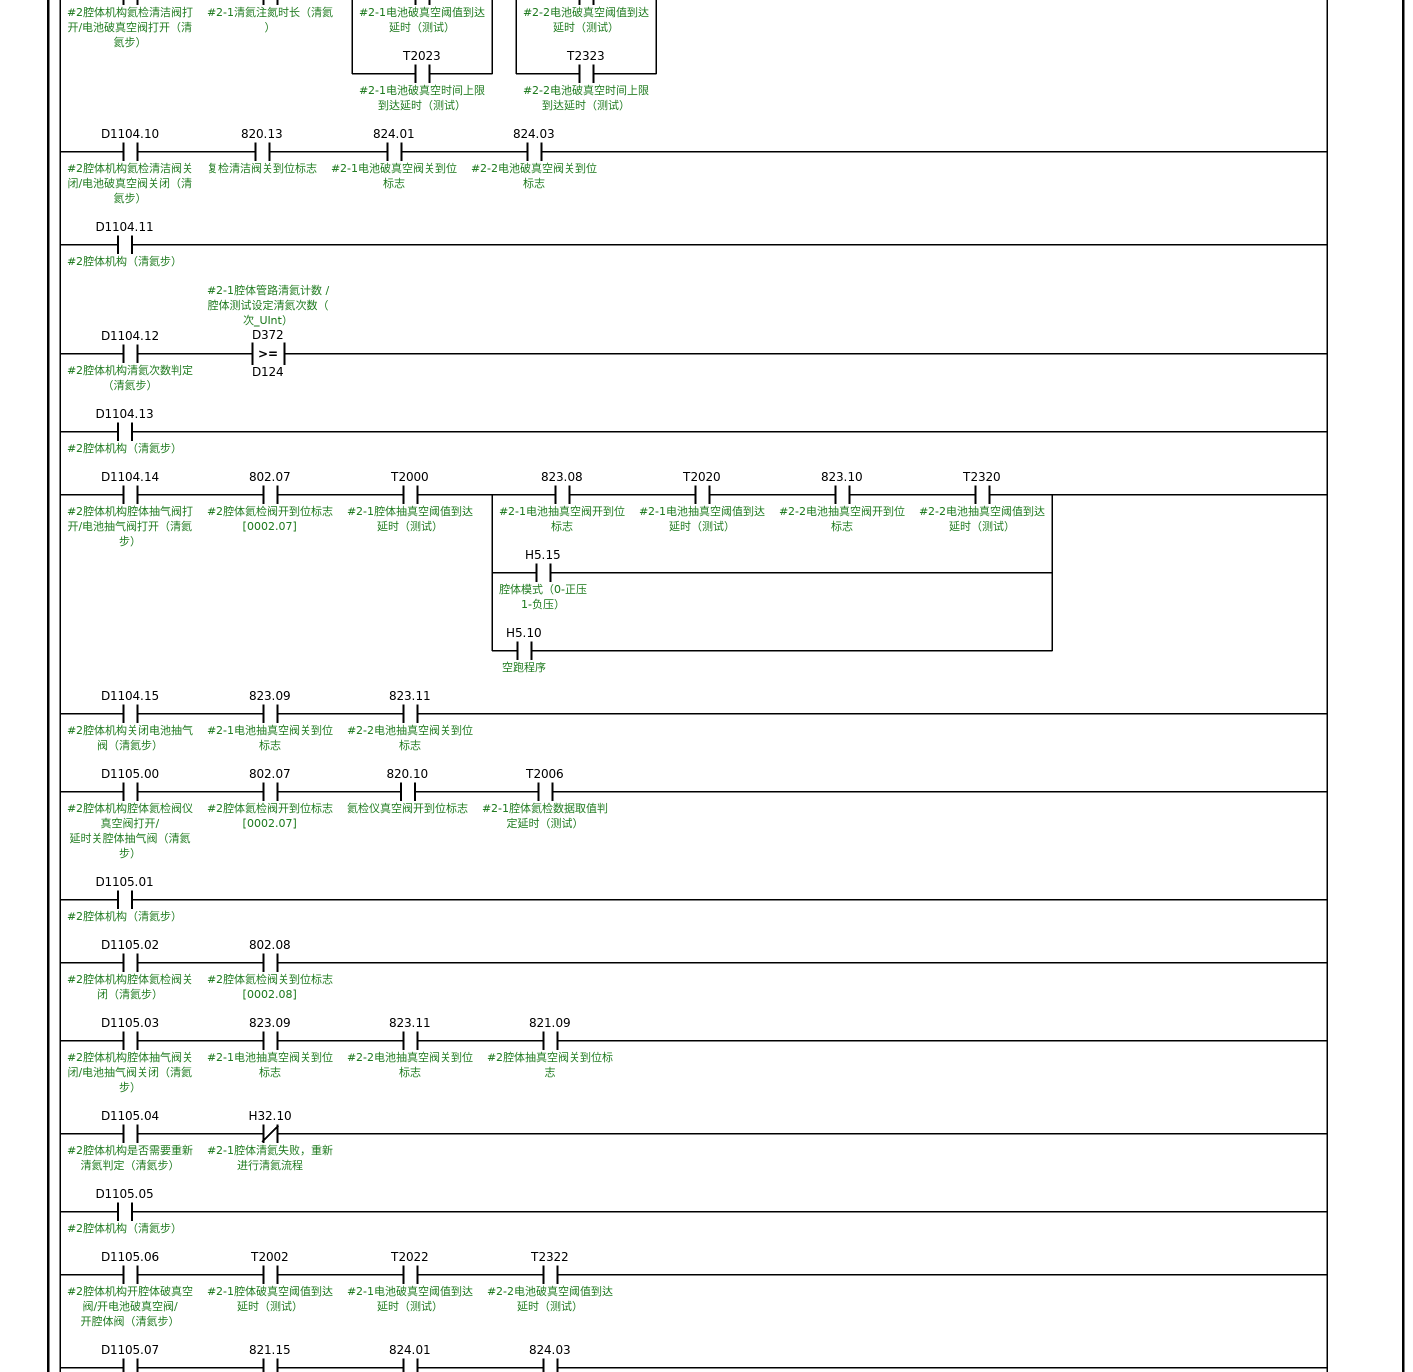

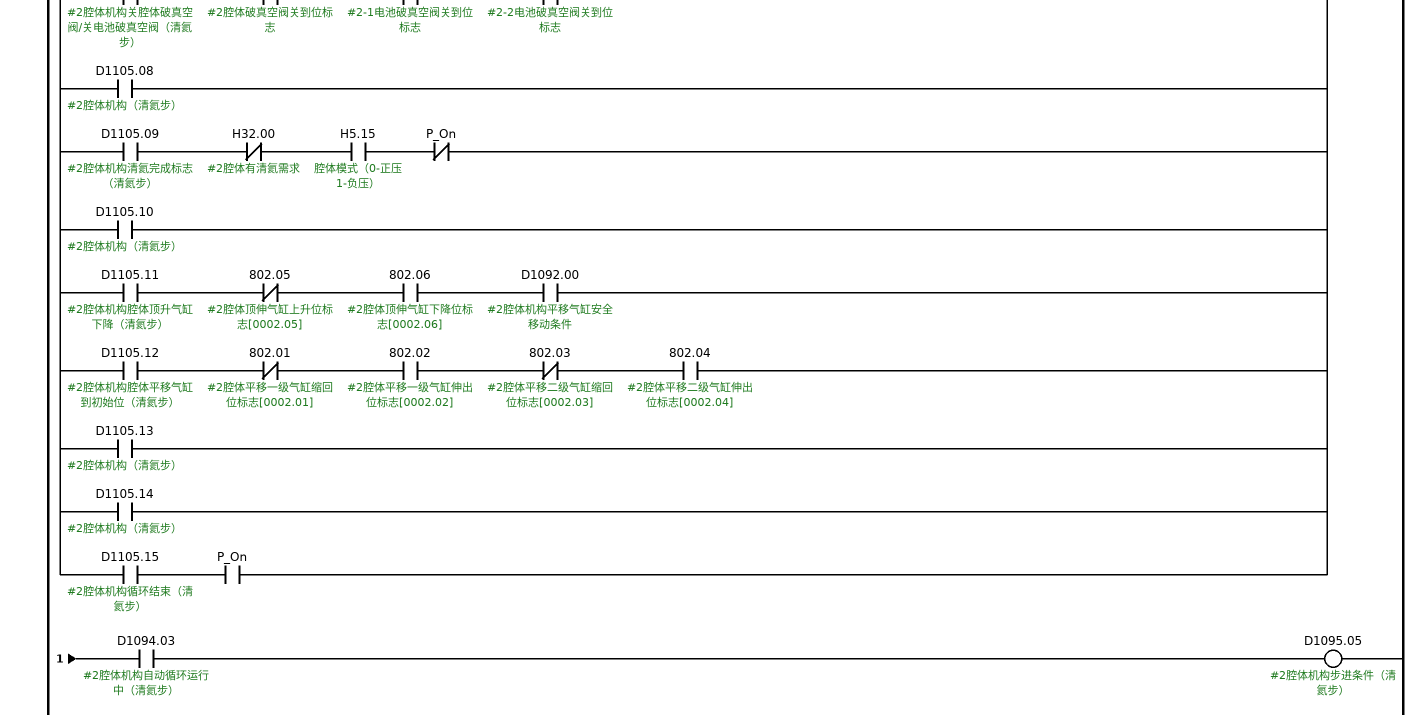
; rung 23
LD D1104.00  ; #2腔体机构自动开始（清氦步）
AND T1556  ; #2腔体机构开始运行延时（清氦步）
LD D1104.01  ; #2腔体机构平移气缸到氦检位/数据初始化（清氦步）
ANDNOT 802.01  ; #2腔体平移一级气缸缩回位标志[0002.01]
AND 802.02  ; #2腔体平移一级气缸伸出位标志[0002.02]
AND 802.03  ; #2腔体平移二级气缸缩回位标志[0002.03]
ANDNOT 802.04  ; #2腔体平移二级气缸伸出位标志[0002.04]
AND T2040  ; #2-1数据初始化延时（清氦）
ORLD
LD D1104.02  ; #2腔体机构腔体顶升气缸上升（清氦步）
AND 802.05  ; #2腔体顶伸气缸上升位标志[0002.05]
ANDNOT 802.06  ; #2腔体顶伸气缸下降位标志[0002.06]
ORLD
LD D1104.03  ; #2腔体机构氦检仪真空阀关闭（清氦步）
AND 820.11  ; 氦检仪真空阀关到位标志
ORLD
LD D1104.04  ; #2腔体机构正压开腔体阀/负压关腔体阀/氦检阀打开  // 负压模式下，复测前的清氦不允许抽电池
LDNOT H5.15  ; 腔体模式（0-正压 1-负压）
LD 821.10  ; #2-1腔体阀开到位标志
AND 821.12  ; #2-2腔体阀开到位标志
LD D1100.11  ; #2腔体机构关闭#2-1腔体阀/清氦判定（自动单检步）
AND 821.10  ; #2-1腔体阀开到位标志
ORLD
LD D1101.07  ; #2腔体机构清氦需求判定（自动单检步）
AND 821.12  ; #2-2腔体阀开到位标志
ORLD
ANDLD
LD H5.15  ; 腔体模式（0-正压 1-负压）
LD D1097.01  ; #2腔体机构清氦需求判定（自动步）
OR D1100.11  ; #2腔体机构关闭#2-1腔体阀/清氦判定（自动单检步）
OR P_On
ANDLD
AND 821.11  ; #2-1腔体阀关到位标志
AND 821.13  ; #2-2腔体阀关到位标志
ORLD
ANDLD
AND D1092.15  ; #2腔体机构腔体抽气阀打开允许
AND D1092.14  ; #2腔体氦检阀打开允许条件
AND 802.07  ; #2腔体氦检阀开到位标志[0002.07]
LD W380.15  ; 氦检仪漏率低于设定值（稳态）
OR H5.02  ; 氦检仪屏蔽
ANDLD
ORLD
OR D1104.05  ; #2腔体机构（清氦步）
LD D1104.06  ; #2腔体机构腔体抽气阀打开/电池抽气阀打开（清氦步）
LD T2000  ; #2-1腔体抽真空阈值到达延时（测试）
OR T2008  ; #2-1腔体抽残气时间上限到达延时（测试）
ANDLD
LD 823.08  ; #2-1电池抽真空阀开到位标志
AND T2020  ; #2-1电池抽真空阈值到达延时（测试）
OR T2021  ; #2-1电池抽真空时间上限到达延时（测试）
LD 823.10  ; #2-2电池抽真空阀开到位标志
AND T2320  ; #2-2电池抽真空阈值到达延时（测试）
OR T2321  ; #2-2电池抽真空时间上限到达延时（测试）
ANDLD
OR H5.15  ; 腔体模式（0-正压 1-负压）
OR H5.10  ; 空跑程序
ANDLD
ORLD
LD D1104.07  ; #2腔体机构腔体抽气阀关闭/电池抽气阀关闭（清氦步）
AND 821.09  ; #2腔体抽真空阀关到位标志
AND 823.09  ; #2-1电池抽真空阀关到位标志
AND 823.11  ; #2-2电池抽真空阀关到位标志
ORLD
OR D1104.08  ; #2腔体机构（清氦步）
LD D1104.09  ; #2腔体机构氦检清洁阀打开/电池破真空阀打开（清氦步）
AND T2041  ; #2-1清氦注氮时长（清氦）
LD T2022  ; #2-1电池破真空阈值到达延时（测试）
OR T2023  ; #2-1电池破真空时间上限到达延时（测试）
ANDLD
LD T2322  ; #2-2电池破真空阈值到达延时（测试）
OR T2323  ; #2-2电池破真空时间上限到达延时（测试）
ANDLD
ORLD
LD D1104.10  ; #2腔体机构氦检清洁阀关闭/电池破真空阀关闭（清氦步）
AND 820.13  ; 复检清洁阀关到位标志
AND 824.01  ; #2-1电池破真空阀关到位标志
AND 824.03  ; #2-2电池破真空阀关到位标志
ORLD
OR D1104.11  ; #2腔体机构（清氦步）
LD D1104.12  ; #2腔体机构清氦次数判定（清氦步）
AND>=(325) D372 D124  ; #2-1腔体管路清氦计数, 腔体测试设定清氦次数（次_UInt）
ORLD
OR D1104.13  ; #2腔体机构（清氦步）
LD D1104.14  ; #2腔体机构腔体抽气阀打开/电池抽气阀打开（清氦步）
AND 802.07  ; #2腔体氦检阀开到位标志[0002.07]
AND T2000  ; #2-1腔体抽真空阈值到达延时（测试）
LD 823.08  ; #2-1电池抽真空阀开到位标志
AND T2020  ; #2-1电池抽真空阈值到达延时（测试）
AND 823.10  ; #2-2电池抽真空阀开到位标志
AND T2320  ; #2-2电池抽真空阈值到达延时（测试）
OR H5.15  ; 腔体模式（0-正压 1-负压）
OR H5.10  ; 空跑程序
ANDLD
ORLD
LD D1104.15  ; #2腔体机构关闭电池抽气阀（清氦步）
AND 823.09  ; #2-1电池抽真空阀关到位标志
AND 823.11  ; #2-2电池抽真空阀关到位标志
ORLD
LD D1105.00  ; #2腔体机构腔体氦检阀仪真空阀打开/延时关腔体抽气阀（清氦步）
AND 802.07  ; #2腔体氦检阀开到位标志[0002.07]
AND 820.10  ; 氦检仪真空阀开到位标志
AND T2006  ; #2-1腔体氦检数据取值判定延时（测试）
ORLD
OR D1105.01  ; #2腔体机构（清氦步）
LD D1105.02  ; #2腔体机构腔体氦检阀关闭（清氦步）
AND 802.08  ; #2腔体氦检阀关到位标志[0002.08]
ORLD
LD D1105.03  ; #2腔体机构腔体抽气阀关闭/电池抽气阀关闭（清氦步）
AND 823.09  ; #2-1电池抽真空阀关到位标志
AND 823.11  ; #2-2电池抽真空阀关到位标志
AND 821.09  ; #2腔体抽真空阀关到位标志
ORLD
LD D1105.04  ; #2腔体机构是否需要重新清氦判定（清氦步）
ANDNOT H32.10  ; #2-1腔体清氦失败，重新进行清氦流程  // 清氦失败，重新进行清氦
ORLD
OR D1105.05  ; #2腔体机构（清氦步）
LD D1105.06  ; #2腔体机构开腔体破真空阀/开电池破真空阀/开腔体阀（清氦步）
AND T2002  ; #2-1腔体破真空阈值到达延时（测试）
AND T2022  ; #2-1电池破真空阈值到达延时（测试）
AND T2322  ; #2-2电池破真空阈值到达延时（测试）
ORLD
LD D1105.07  ; #2腔体机构关腔体破真空阀/关电池破真空阀（清氦步）
AND 821.15  ; #2腔体破真空阀关到位标志
AND 824.01  ; #2-1电池破真空阀关到位标志
AND 824.03  ; #2-2电池破真空阀关到位标志
ORLD
OR D1105.08  ; #2腔体机构（清氦步）
LD D1105.09  ; #2腔体机构清氦完成标志（清氦步）  // 正压腔体是待料清氦，需跳转回测试步序
ANDNOT H32.00  ; #2腔体有清氦需求
AND H5.15  ; 腔体模式（0-正压 1-负压）
ANDNOT P_On
ORLD
OR D1105.10  ; #2腔体机构（清氦步）
LD D1105.11  ; #2腔体机构腔体顶升气缸下降（清氦步）
ANDNOT 802.05  ; #2腔体顶伸气缸上升位标志[0002.05]
AND 802.06  ; #2腔体顶伸气缸下降位标志[0002.06]
AND D1092.00  ; #2腔体机构平移气缸安全移动条件
ORLD
LD D1105.12  ; #2腔体机构腔体平移气缸到初始位（清氦步）
ANDNOT 802.01  ; #2腔体平移一级气缸缩回位标志[0002.01]
AND 802.02  ; #2腔体平移一级气缸伸出位标志[0002.02]
ANDNOT 802.03  ; #2腔体平移二级气缸缩回位标志[0002.03]
AND 802.04  ; #2腔体平移二级气缸伸出位标志[0002.04]
ORLD
OR D1105.13  ; #2腔体机构（清氦步）
OR D1105.14  ; #2腔体机构（清氦步）
LD D1105.15  ; #2腔体机构循环结束（清氦步）
AND P_On
ORLD
AND D1094.03  ; #2腔体机构自动循环运行中（清氦步）
OUT D1095.05  ; #2腔体机构步进条件（清氦步）

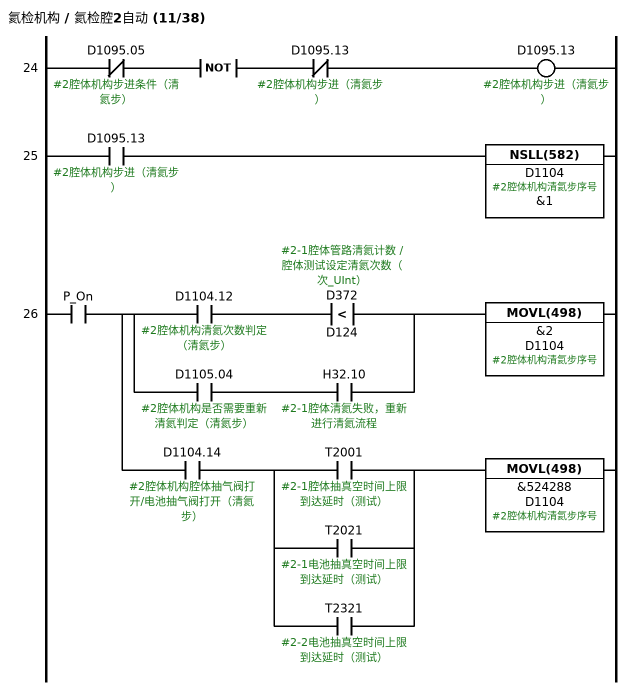
; rung 24
LDNOT D1095.05  ; #2腔体机构步进条件（清氦步）
NOT(520)
ANDNOT D1095.13  ; #2腔体机构步进（清氦步）
OUT D1095.13  ; #2腔体机构步进（清氦步）
; rung 25
LD D1095.13  ; #2腔体机构步进（清氦步）
NSLL(582) D1104 &1  ; #2腔体机构清氦步序号
; rung 26
LD P_On
OUT TR0
LD D1104.12  ; #2腔体机构清氦次数判定（清氦步）
AND<(310) D372 D124  ; #2-1腔体管路清氦计数, 腔体测试设定清氦次数（次_UInt）
LD D1105.04  ; #2腔体机构是否需要重新清氦判定（清氦步）
AND H32.10  ; #2-1腔体清氦失败，重新进行清氦流程  // 清氦失败，重新进行清氦
ORLD
ANDLD
MOVL(498) &2 D1104  ; #2腔体机构清氦步序号
LD TR0
AND D1104.14  ; #2腔体机构腔体抽气阀打开/电池抽气阀打开（清氦步）
LD T2001  ; #2-1腔体抽真空时间上限到达延时（测试）
OR T2021  ; #2-1电池抽真空时间上限到达延时（测试）
OR T2321  ; #2-2电池抽真空时间上限到达延时（测试）
ANDLD
MOVL(498) &524288 D1104  ; #2腔体机构清氦步序号  // 清氦过程腔体或电池抽气上限达到，均直接判定清氦完成，不进入氦检步序（跳转至D1075.03）

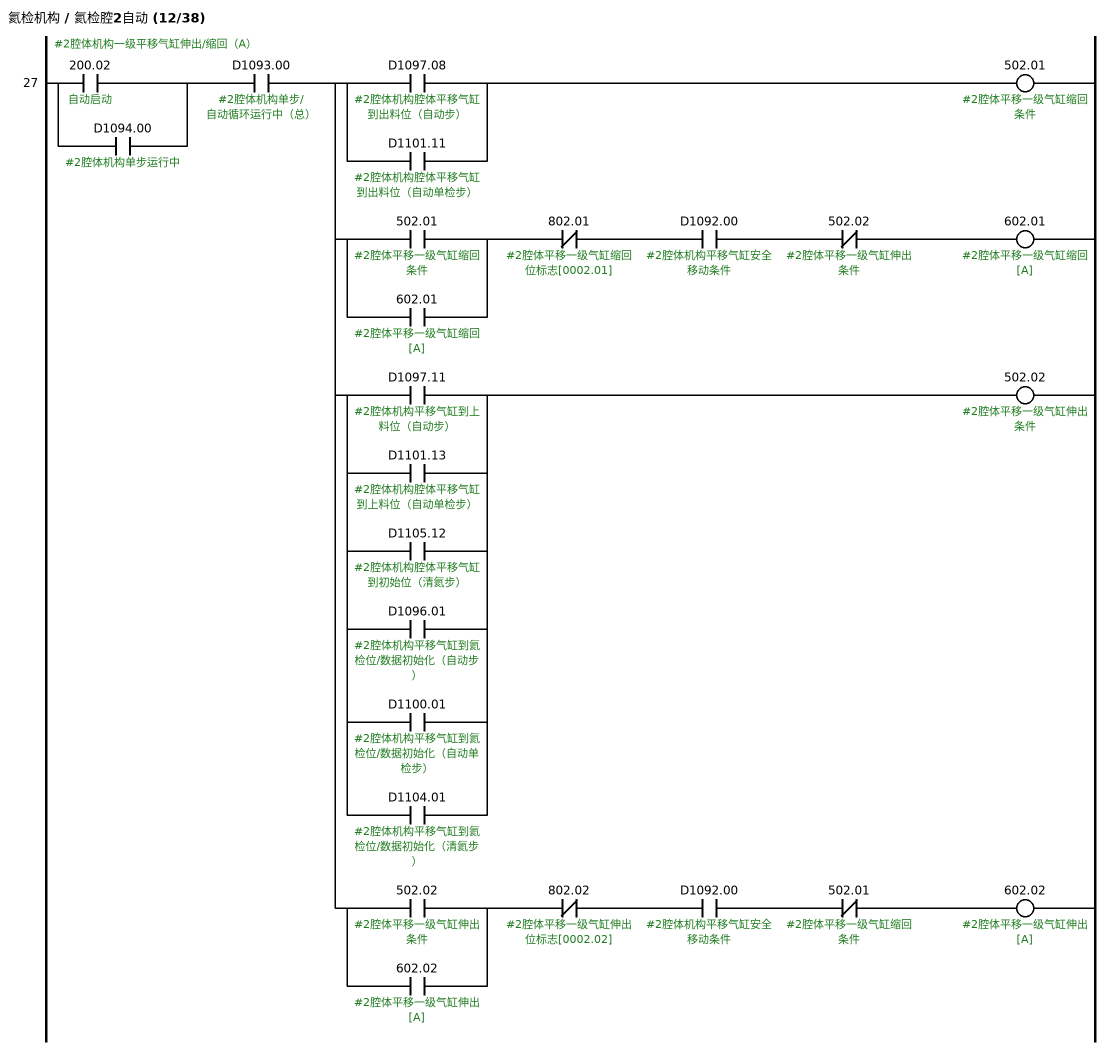
; rung 27: #2腔体机构一级平移气缸伸出/缩回（A）
LD 200.02  ; 自动启动
OR D1094.00  ; #2腔体机构单步运行中
AND D1093.00  ; #2腔体机构单步/自动循环运行中（总）
OUT TR0
LD D1097.08  ; #2腔体机构腔体平移气缸到出料位（自动步）
OR D1101.11  ; #2腔体机构腔体平移气缸到出料位（自动单检步）
ANDLD
OUT 502.01  ; #2腔体平移一级气缸缩回条件
LD TR0
LD 502.01  ; #2腔体平移一级气缸缩回条件
OR 602.01  ; #2腔体平移一级气缸缩回[A]
ANDLD
ANDNOT 802.01  ; #2腔体平移一级气缸缩回位标志[0002.01]
AND D1092.00  ; #2腔体机构平移气缸安全移动条件
ANDNOT 502.02  ; #2腔体平移一级气缸伸出条件
OUT 602.01  ; #2腔体平移一级气缸缩回[A]
LD TR0
LD D1097.11  ; #2腔体机构平移气缸到上料位（自动步）
OR D1101.13  ; #2腔体机构腔体平移气缸到上料位（自动单检步）
OR D1105.12  ; #2腔体机构腔体平移气缸到初始位（清氦步）
OR D1096.01  ; #2腔体机构平移气缸到氦检位/数据初始化（自动步）
OR D1100.01  ; #2腔体机构平移气缸到氦检位/数据初始化（自动单检步）
OR D1104.01  ; #2腔体机构平移气缸到氦检位/数据初始化（清氦步）
ANDLD
OUT 502.02  ; #2腔体平移一级气缸伸出条件
LD TR0
LD 502.02  ; #2腔体平移一级气缸伸出条件
OR 602.02  ; #2腔体平移一级气缸伸出[A]
ANDLD
ANDNOT 802.02  ; #2腔体平移一级气缸伸出位标志[0002.02]
AND D1092.00  ; #2腔体机构平移气缸安全移动条件
ANDNOT 502.01  ; #2腔体平移一级气缸缩回条件
OUT 602.02  ; #2腔体平移一级气缸伸出[A]

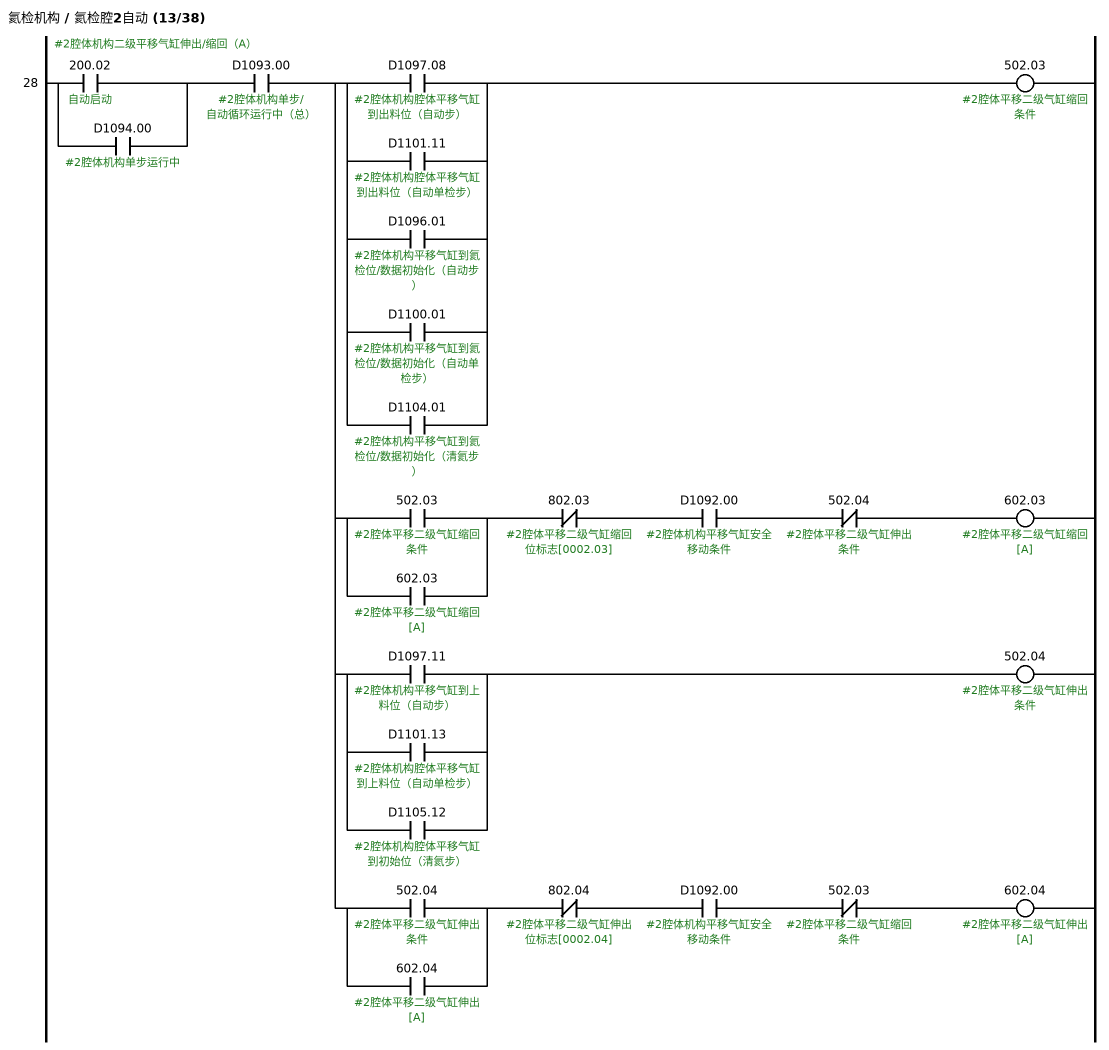
; rung 28: #2腔体机构二级平移气缸伸出/缩回（A）
LD 200.02  ; 自动启动
OR D1094.00  ; #2腔体机构单步运行中
AND D1093.00  ; #2腔体机构单步/自动循环运行中（总）
OUT TR0
LD D1097.08  ; #2腔体机构腔体平移气缸到出料位（自动步）
OR D1101.11  ; #2腔体机构腔体平移气缸到出料位（自动单检步）
OR D1096.01  ; #2腔体机构平移气缸到氦检位/数据初始化（自动步）
OR D1100.01  ; #2腔体机构平移气缸到氦检位/数据初始化（自动单检步）
OR D1104.01  ; #2腔体机构平移气缸到氦检位/数据初始化（清氦步）
ANDLD
OUT 502.03  ; #2腔体平移二级气缸缩回条件
LD TR0
LD 502.03  ; #2腔体平移二级气缸缩回条件
OR 602.03  ; #2腔体平移二级气缸缩回[A]
ANDLD
ANDNOT 802.03  ; #2腔体平移二级气缸缩回位标志[0002.03]
AND D1092.00  ; #2腔体机构平移气缸安全移动条件
ANDNOT 502.04  ; #2腔体平移二级气缸伸出条件
OUT 602.03  ; #2腔体平移二级气缸缩回[A]
LD TR0
LD D1097.11  ; #2腔体机构平移气缸到上料位（自动步）
OR D1101.13  ; #2腔体机构腔体平移气缸到上料位（自动单检步）
OR D1105.12  ; #2腔体机构腔体平移气缸到初始位（清氦步）
ANDLD
OUT 502.04  ; #2腔体平移二级气缸伸出条件
LD TR0
LD 502.04  ; #2腔体平移二级气缸伸出条件
OR 602.04  ; #2腔体平移二级气缸伸出[A]
ANDLD
ANDNOT 802.04  ; #2腔体平移二级气缸伸出位标志[0002.04]
AND D1092.00  ; #2腔体机构平移气缸安全移动条件
ANDNOT 502.03  ; #2腔体平移二级气缸缩回条件
OUT 602.04  ; #2腔体平移二级气缸伸出[A]

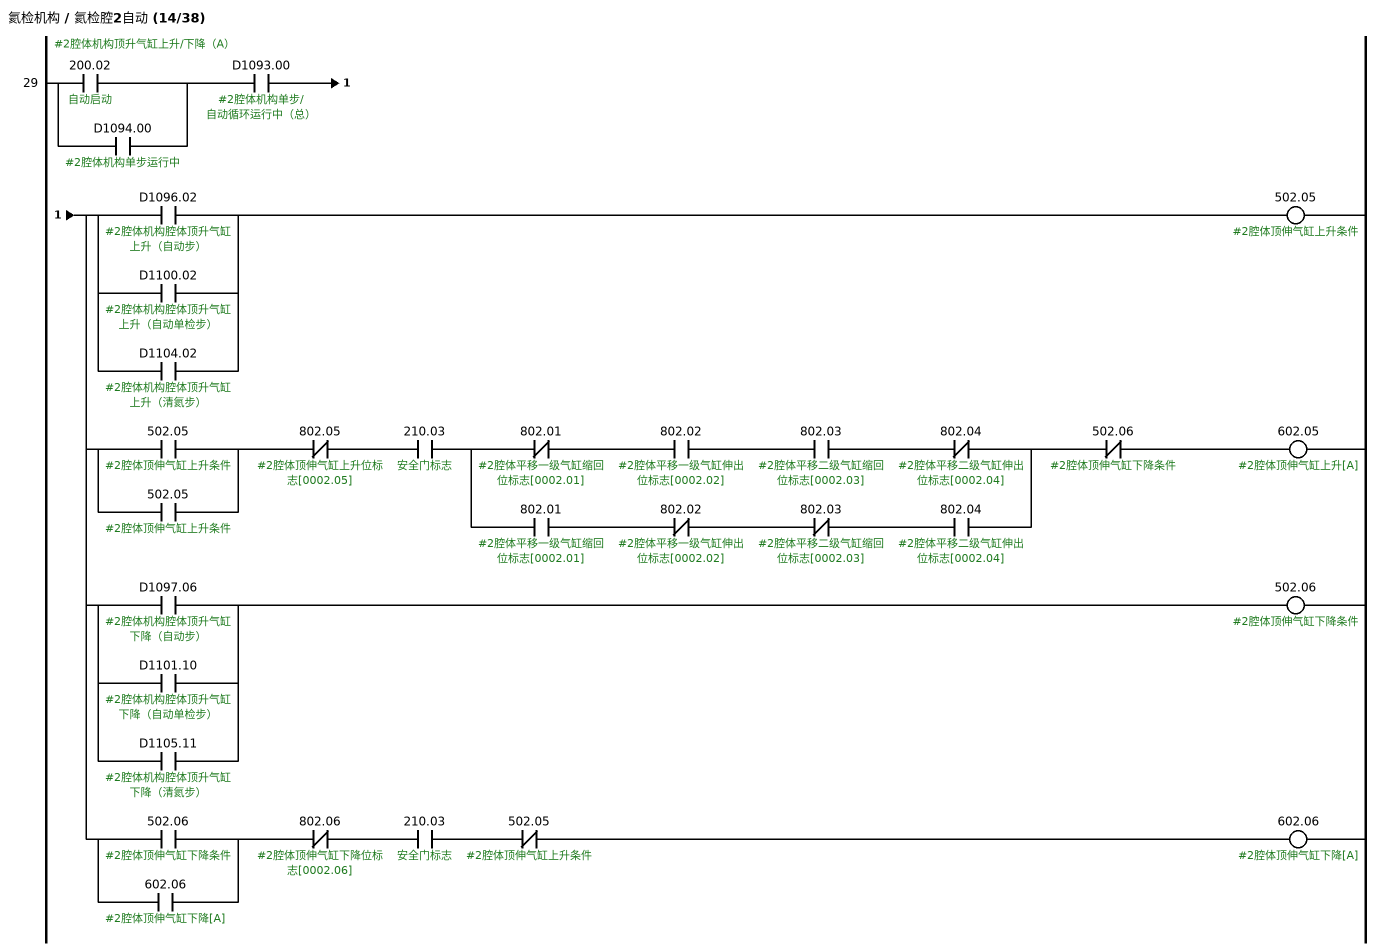
; rung 29: #2腔体机构顶升气缸上升/下降（A）
LD 200.02  ; 自动启动
OR D1094.00  ; #2腔体机构单步运行中
AND D1093.00  ; #2腔体机构单步/自动循环运行中（总）
OUT TR0
LD D1096.02  ; #2腔体机构腔体顶升气缸上升（自动步）
OR D1100.02  ; #2腔体机构腔体顶升气缸上升（自动单检步）
OR D1104.02  ; #2腔体机构腔体顶升气缸上升（清氦步）
ANDLD
OUT 502.05  ; #2腔体顶伸气缸上升条件
LD TR0
LD 502.05  ; #2腔体顶伸气缸上升条件
OR 502.05  ; #2腔体顶伸气缸上升条件
ANDLD
ANDNOT 802.05  ; #2腔体顶伸气缸上升位标志[0002.05]
AND 210.03  ; 安全门标志
LDNOT 802.01  ; #2腔体平移一级气缸缩回位标志[0002.01]
AND 802.02  ; #2腔体平移一级气缸伸出位标志[0002.02]
AND 802.03  ; #2腔体平移二级气缸缩回位标志[0002.03]
ANDNOT 802.04  ; #2腔体平移二级气缸伸出位标志[0002.04]
LD 802.01  ; #2腔体平移一级气缸缩回位标志[0002.01]
ANDNOT 802.02  ; #2腔体平移一级气缸伸出位标志[0002.02]
ANDNOT 802.03  ; #2腔体平移二级气缸缩回位标志[0002.03]
AND 802.04  ; #2腔体平移二级气缸伸出位标志[0002.04]
ORLD
ANDLD
ANDNOT 502.06  ; #2腔体顶伸气缸下降条件
OUT 602.05  ; #2腔体顶伸气缸上升[A]
LD TR0
LD D1097.06  ; #2腔体机构腔体顶升气缸下降（自动步）
OR D1101.10  ; #2腔体机构腔体顶升气缸下降（自动单检步）
OR D1105.11  ; #2腔体机构腔体顶升气缸下降（清氦步）
ANDLD
OUT 502.06  ; #2腔体顶伸气缸下降条件
LD TR0
LD 502.06  ; #2腔体顶伸气缸下降条件
OR 602.06  ; #2腔体顶伸气缸下降[A]
ANDLD
ANDNOT 802.06  ; #2腔体顶伸气缸下降位标志[0002.06]
AND 210.03  ; 安全门标志
ANDNOT 502.05  ; #2腔体顶伸气缸上升条件
OUT 602.06  ; #2腔体顶伸气缸下降[A]

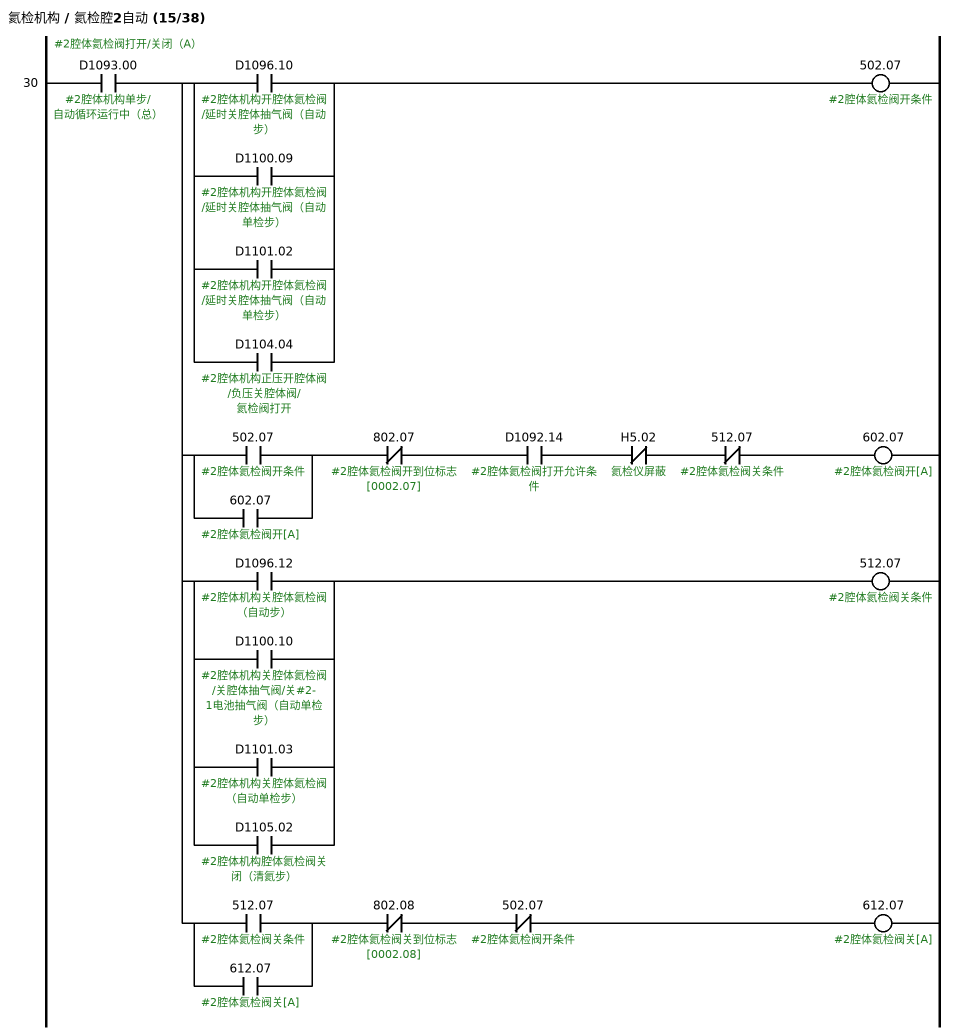
; rung 30: #2腔体氦检阀打开/关闭（A）
LD D1093.00  ; #2腔体机构单步/自动循环运行中（总）
OUT TR0
LD D1096.10  ; #2腔体机构开腔体氦检阀/延时关腔体抽气阀（自动步）
OR D1100.09  ; #2腔体机构开腔体氦检阀/延时关腔体抽气阀（自动单检步）
OR D1101.02  ; #2腔体机构开腔体氦检阀/延时关腔体抽气阀（自动单检步）
OR D1104.04  ; #2腔体机构正压开腔体阀/负压关腔体阀/氦检阀打开
ANDLD
OUT 502.07  ; #2腔体氦检阀开条件
LD TR0
LD 502.07  ; #2腔体氦检阀开条件
OR 602.07  ; #2腔体氦检阀开[A]
ANDLD
ANDNOT 802.07  ; #2腔体氦检阀开到位标志[0002.07]
AND D1092.14  ; #2腔体氦检阀打开允许条件
ANDNOT H5.02  ; 氦检仪屏蔽
ANDNOT 512.07  ; #2腔体氦检阀关条件
OUT 602.07  ; #2腔体氦检阀开[A]
LD TR0
LD D1096.12  ; #2腔体机构关腔体氦检阀（自动步）
OR D1100.10  ; #2腔体机构关腔体氦检阀/关腔体抽气阀/关#2-1电池抽气阀（自动单检步）
OR D1101.03  ; #2腔体机构关腔体氦检阀（自动单检步）
OR D1105.02  ; #2腔体机构腔体氦检阀关闭（清氦步）
ANDLD
OUT 512.07  ; #2腔体氦检阀关条件
LD TR0
LD 512.07  ; #2腔体氦检阀关条件
OR 612.07  ; #2腔体氦检阀关[A]
ANDLD
ANDNOT 802.08  ; #2腔体氦检阀关到位标志[0002.08]
ANDNOT 502.07  ; #2腔体氦检阀开条件
OUT 612.07  ; #2腔体氦检阀关[A]

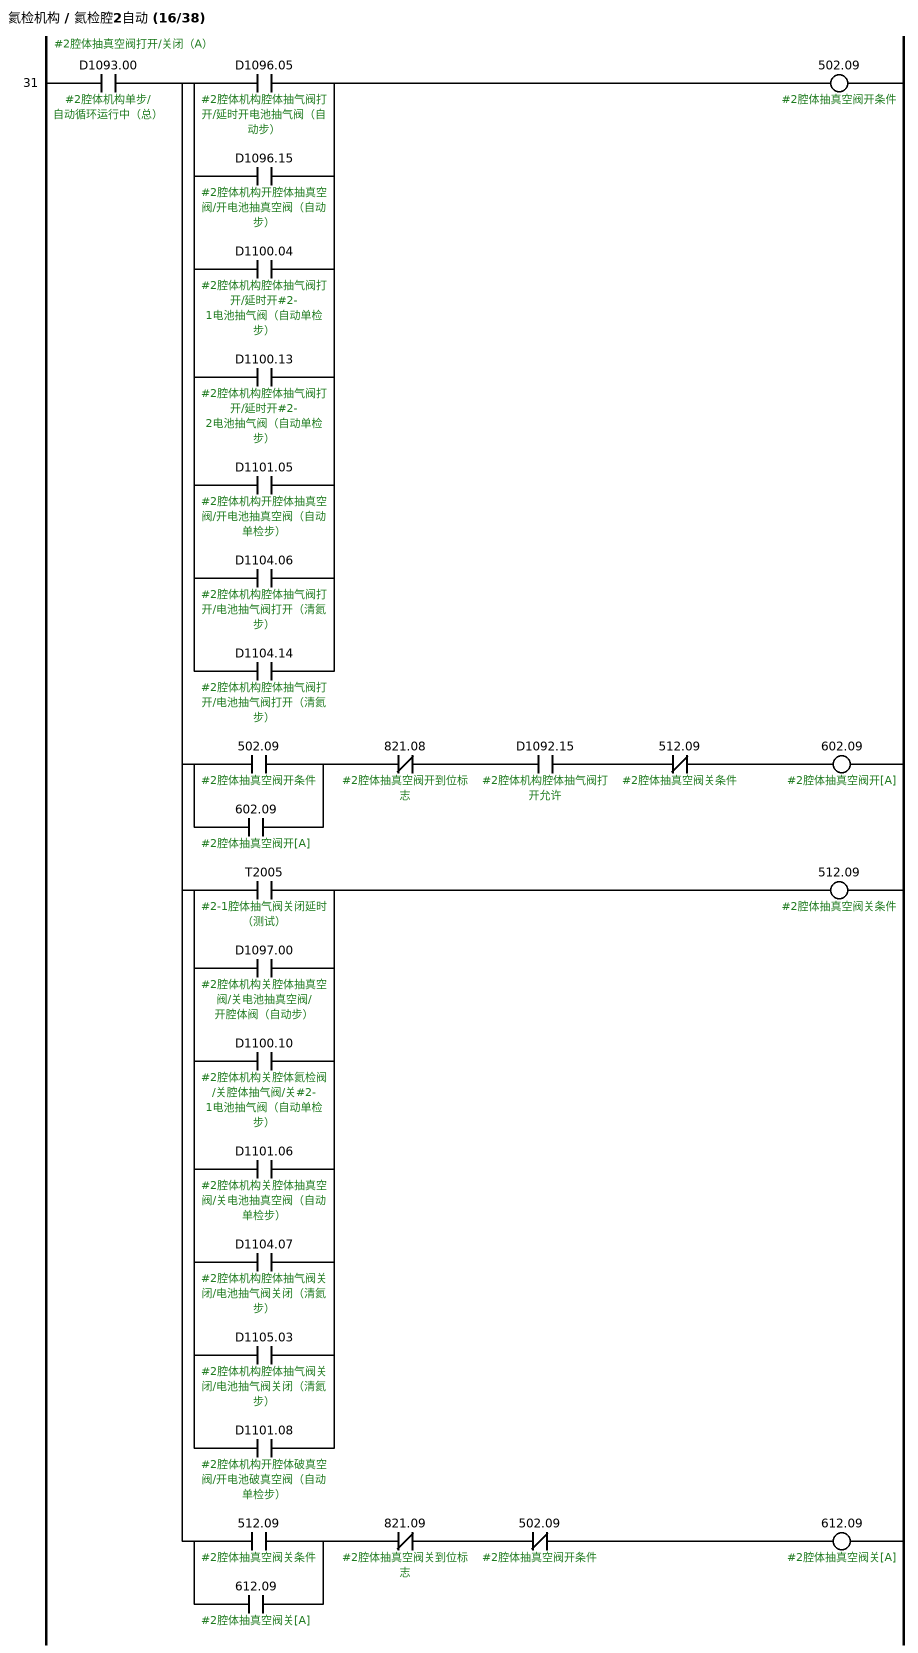
; rung 31: #2腔体抽真空阀打开/关闭（A）
LD D1093.00  ; #2腔体机构单步/自动循环运行中（总）
OUT TR0
LD D1096.05  ; #2腔体机构腔体抽气阀打开/延时开电池抽气阀（自动步）
OR D1096.15  ; #2腔体机构开腔体抽真空阀/开电池抽真空阀（自动步）
OR D1100.04  ; #2腔体机构腔体抽气阀打开/延时开#2-1电池抽气阀（自动单检步）
OR D1100.13  ; #2腔体机构腔体抽气阀打开/延时开#2-2电池抽气阀（自动单检步）
OR D1101.05  ; #2腔体机构开腔体抽真空阀/开电池抽真空阀（自动单检步）
OR D1104.06  ; #2腔体机构腔体抽气阀打开/电池抽气阀打开（清氦步）
OR D1104.14  ; #2腔体机构腔体抽气阀打开/电池抽气阀打开（清氦步）
ANDLD
OUT 502.09  ; #2腔体抽真空阀开条件
LD TR0
LD 502.09  ; #2腔体抽真空阀开条件
OR 602.09  ; #2腔体抽真空阀开[A]
ANDLD
ANDNOT 821.08  ; #2腔体抽真空阀开到位标志
AND D1092.15  ; #2腔体机构腔体抽气阀打开允许
ANDNOT 512.09  ; #2腔体抽真空阀关条件
OUT 602.09  ; #2腔体抽真空阀开[A]
LD TR0
LD T2005  ; #2-1腔体抽气阀关闭延时（测试）
OR D1097.00  ; #2腔体机构关腔体抽真空阀/关电池抽真空阀/开腔体阀（自动步）
OR D1100.10  ; #2腔体机构关腔体氦检阀/关腔体抽气阀/关#2-1电池抽气阀（自动单检步）
OR D1101.06  ; #2腔体机构关腔体抽真空阀/关电池抽真空阀（自动单检步）
OR D1104.07  ; #2腔体机构腔体抽气阀关闭/电池抽气阀关闭（清氦步）
OR D1105.03  ; #2腔体机构腔体抽气阀关闭/电池抽气阀关闭（清氦步）
OR D1101.08  ; #2腔体机构开腔体破真空阀/开电池破真空阀（自动单检步）
ANDLD
OUT 512.09  ; #2腔体抽真空阀关条件
LD TR0
LD 512.09  ; #2腔体抽真空阀关条件
OR 612.09  ; #2腔体抽真空阀关[A]
ANDLD
ANDNOT 821.09  ; #2腔体抽真空阀关到位标志
ANDNOT 502.09  ; #2腔体抽真空阀开条件
OUT 612.09  ; #2腔体抽真空阀关[A]

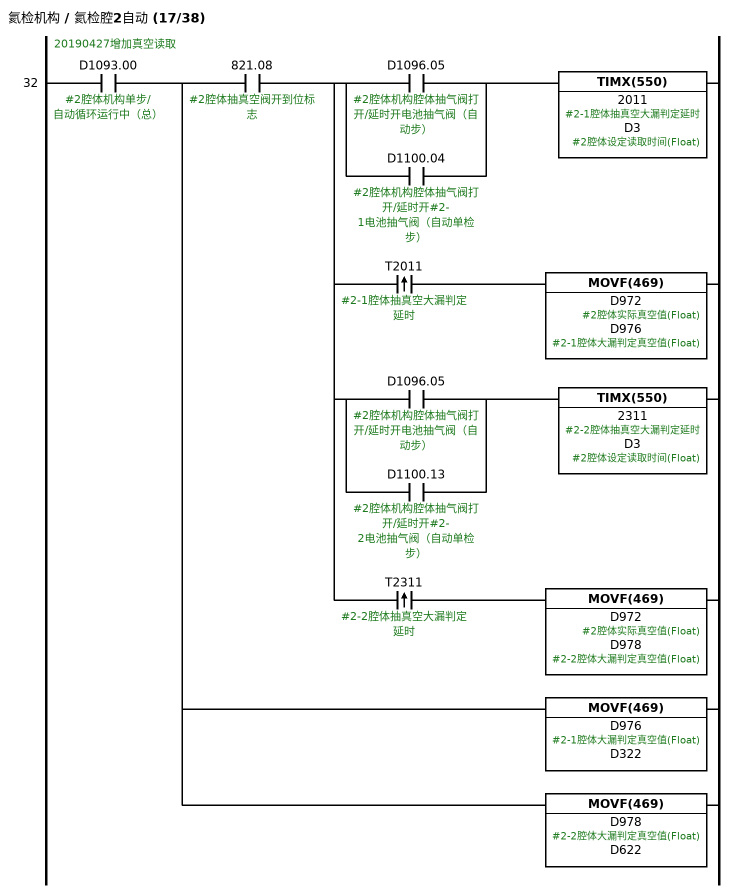
; rung 32: 20190427增加真空读取
LD D1093.00  ; #2腔体机构单步/自动循环运行中（总）
OUT TR0
AND 821.08  ; #2腔体抽真空阀开到位标志
OUT TR1
LD D1096.05  ; #2腔体机构腔体抽气阀打开/延时开电池抽气阀（自动步）
OR D1100.04  ; #2腔体机构腔体抽气阀打开/延时开#2-1电池抽气阀（自动单检步）
ANDLD
TIMX(550) 2011 D3  ; #2腔体设定读取时间(Float), #2-1腔体抽真空大漏判定延时
LD TR1
@AND T2011  ; #2-1腔体抽真空大漏判定延时
MOVF(469) D972 D976  ; #2腔体实际真空值(Float), #2-1腔体大漏判定真空值(Float)
LD TR1
LD D1096.05  ; #2腔体机构腔体抽气阀打开/延时开电池抽气阀（自动步）
OR D1100.13  ; #2腔体机构腔体抽气阀打开/延时开#2-2电池抽气阀（自动单检步）
ANDLD
TIMX(550) 2311 D3  ; #2腔体设定读取时间(Float), #2-2腔体抽真空大漏判定延时
LD TR1
@AND T2311  ; #2-2腔体抽真空大漏判定延时
MOVF(469) D972 D978  ; #2腔体实际真空值(Float), #2-2腔体大漏判定真空值(Float)
LD TR0
MOVF(469) D976 D322  ; #2-1腔体大漏判定真空值(Float)
MOVF(469) D978 D622  ; #2-2腔体大漏判定真空值(Float)

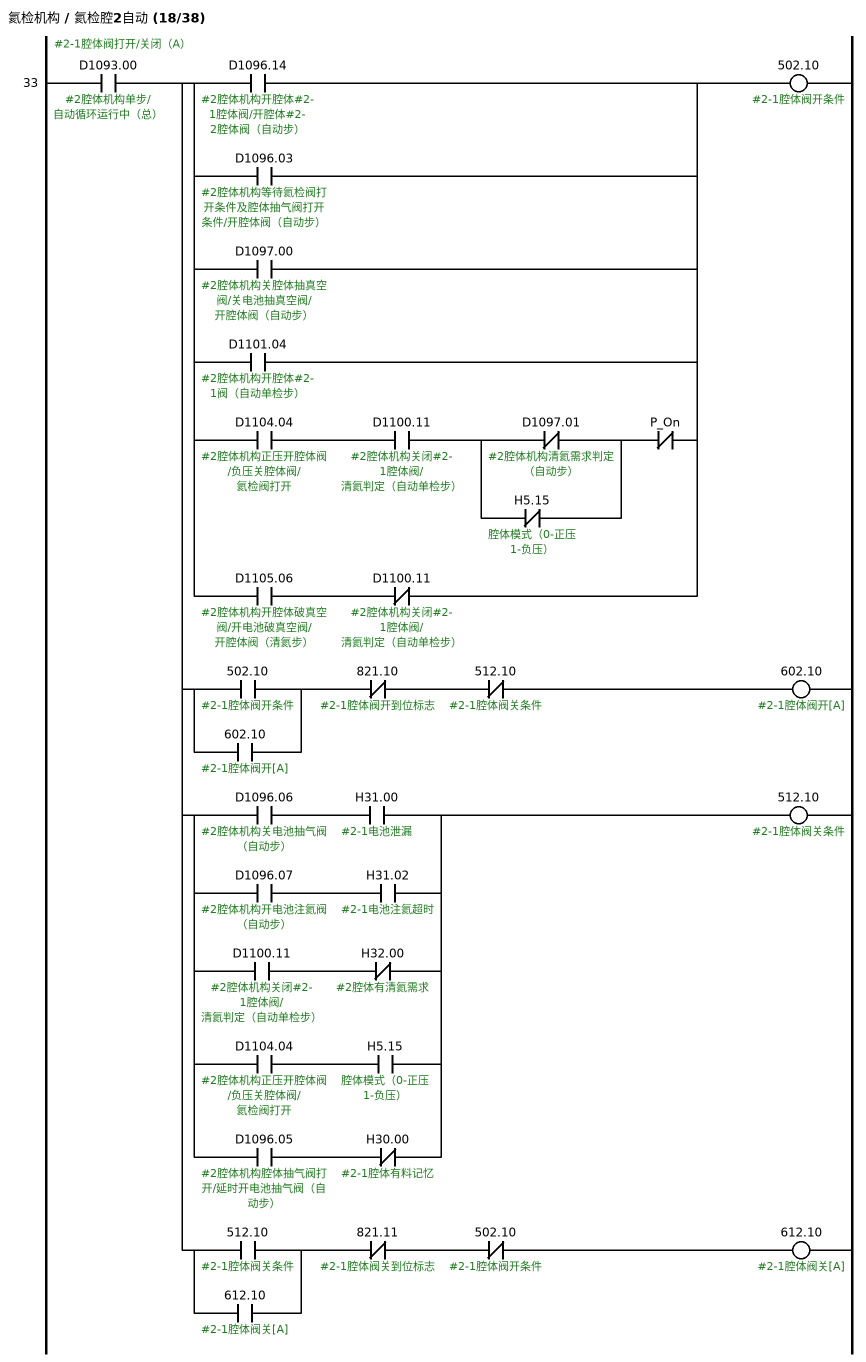
; rung 33: #2-1腔体阀打开/关闭（A）
LD D1093.00  ; #2腔体机构单步/自动循环运行中（总）
OUT TR0
LD D1096.14  ; #2腔体机构开腔体#2-1腔体阀/开腔体#2-2腔体阀（自动步）
OR D1096.03  ; #2腔体机构等待氦检阀打开条件及腔体抽气阀打开条件/开腔体阀（自动步）
OR D1097.00  ; #2腔体机构关腔体抽真空阀/关电池抽真空阀/开腔体阀（自动步）
OR D1101.04  ; #2腔体机构开腔体#2-1阀（自动单检步）
LD D1104.04  ; #2腔体机构正压开腔体阀/负压关腔体阀/氦检阀打开
AND D1100.11  ; #2腔体机构关闭#2-1腔体阀/清氦判定（自动单检步）
LDNOT D1097.01  ; #2腔体机构清氦需求判定（自动步）
ORNOT H5.15  ; 腔体模式（0-正压 1-负压）
ANDLD
ANDNOT P_On
ORLD
LD D1105.06  ; #2腔体机构开腔体破真空阀/开电池破真空阀/开腔体阀（清氦步）
ANDNOT D1100.11  ; #2腔体机构关闭#2-1腔体阀/清氦判定（自动单检步）
ORLD
ANDLD
OUT 502.10  ; #2-1腔体阀开条件
LD TR0
LD 502.10  ; #2-1腔体阀开条件
OR 602.10  ; #2-1腔体阀开[A]
ANDLD
ANDNOT 821.10  ; #2-1腔体阀开到位标志
ANDNOT 512.10  ; #2-1腔体阀关条件
OUT 602.10  ; #2-1腔体阀开[A]
LD TR0
LD D1096.06  ; #2腔体机构关电池抽气阀（自动步）
AND H31.00  ; #2-1电池泄漏
LD D1096.07  ; #2腔体机构开电池注氦阀（自动步）
AND H31.02  ; #2-1电池注氦超时
ORLD
LD D1100.11  ; #2腔体机构关闭#2-1腔体阀/清氦判定（自动单检步）
ANDNOT H32.00  ; #2腔体有清氦需求
ORLD
LD D1104.04  ; #2腔体机构正压开腔体阀/负压关腔体阀/氦检阀打开
AND H5.15  ; 腔体模式（0-正压 1-负压）
ORLD
LD D1096.05  ; #2腔体机构腔体抽气阀打开/延时开电池抽气阀（自动步）  // #1-1无料时不测试
ANDNOT H30.00  ; #2-1腔体有料记忆
ORLD
ANDLD
OUT 512.10  ; #2-1腔体阀关条件
LD TR0
LD 512.10  ; #2-1腔体阀关条件
OR 612.10  ; #2-1腔体阀关[A]
ANDLD
ANDNOT 821.11  ; #2-1腔体阀关到位标志
ANDNOT 502.10  ; #2-1腔体阀开条件
OUT 612.10  ; #2-1腔体阀关[A]

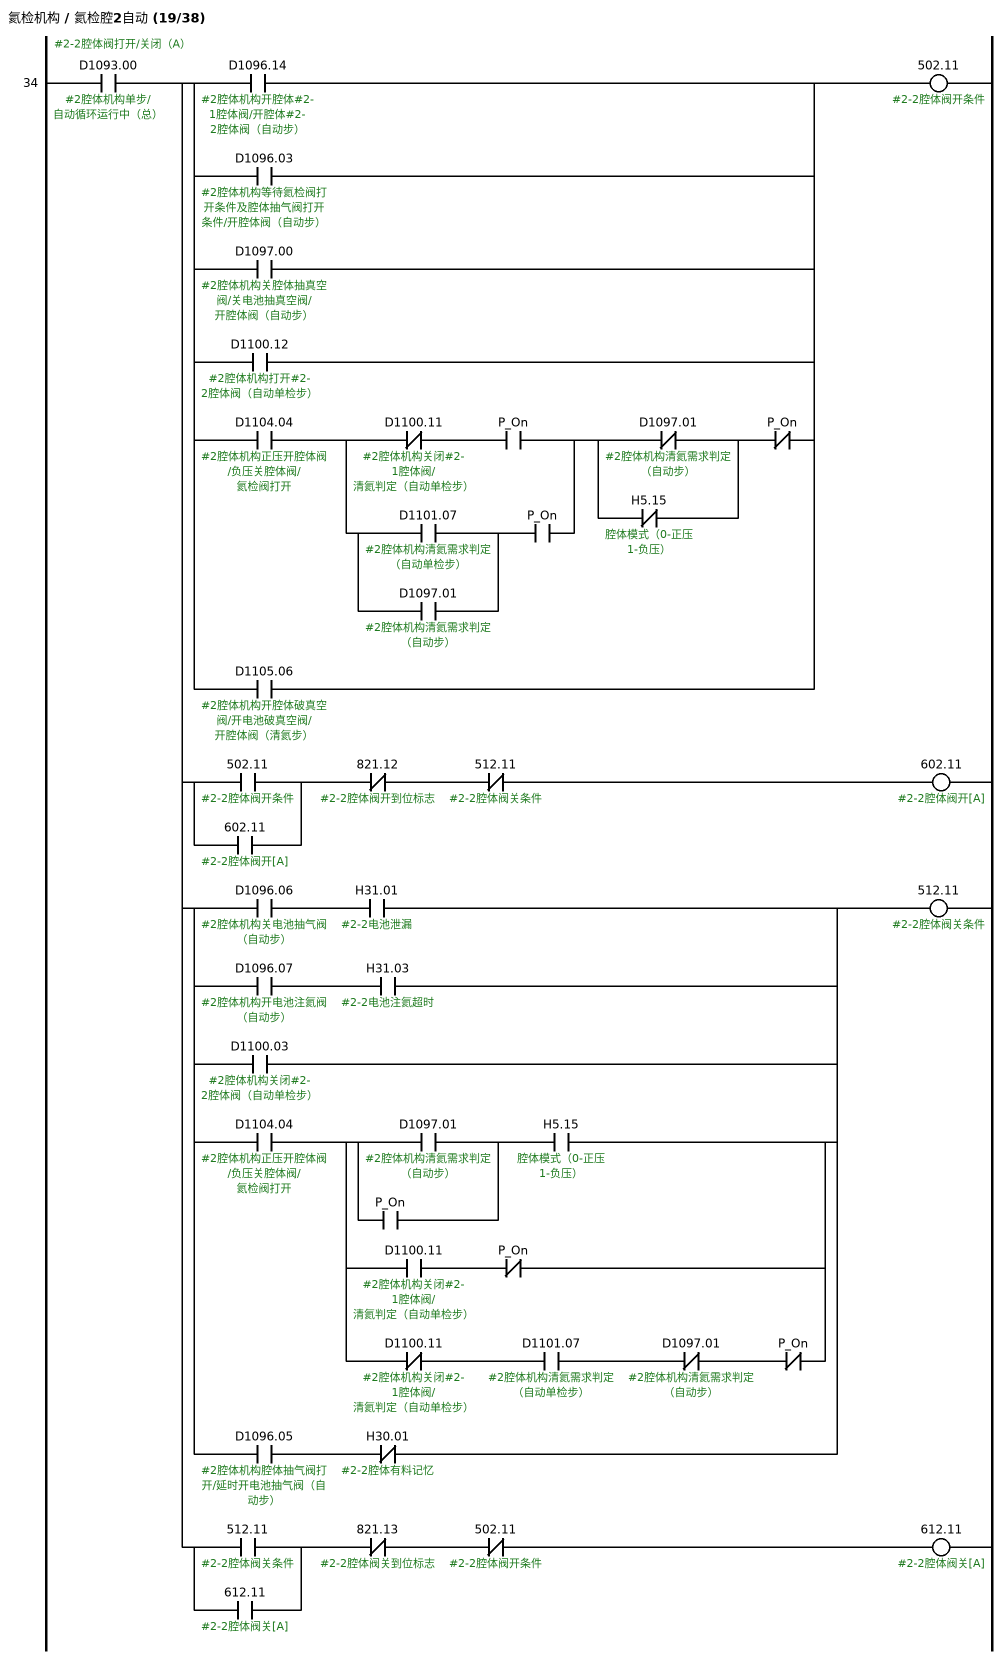
; rung 34: #2-2腔体阀打开/关闭（A）
LD D1093.00  ; #2腔体机构单步/自动循环运行中（总）
OUT TR0
LD D1096.14  ; #2腔体机构开腔体#2-1腔体阀/开腔体#2-2腔体阀（自动步）
OR D1096.03  ; #2腔体机构等待氦检阀打开条件及腔体抽气阀打开条件/开腔体阀（自动步）
OR D1097.00  ; #2腔体机构关腔体抽真空阀/关电池抽真空阀/开腔体阀（自动步）
OR D1100.12  ; #2腔体机构打开#2-2腔体阀（自动单检步）
LD D1104.04  ; #2腔体机构正压开腔体阀/负压关腔体阀/氦检阀打开
LDNOT D1100.11  ; #2腔体机构关闭#2-1腔体阀/清氦判定（自动单检步）
AND P_On
LD D1101.07  ; #2腔体机构清氦需求判定（自动单检步）
OR D1097.01  ; #2腔体机构清氦需求判定（自动步）
AND P_On
ORLD
ANDLD
LDNOT D1097.01  ; #2腔体机构清氦需求判定（自动步）
ORNOT H5.15  ; 腔体模式（0-正压 1-负压）
ANDLD
ANDNOT P_On
ORLD
OR D1105.06  ; #2腔体机构开腔体破真空阀/开电池破真空阀/开腔体阀（清氦步）
ANDLD
OUT 502.11  ; #2-2腔体阀开条件
LD TR0
LD 502.11  ; #2-2腔体阀开条件
OR 602.11  ; #2-2腔体阀开[A]
ANDLD
ANDNOT 821.12  ; #2-2腔体阀开到位标志
ANDNOT 512.11  ; #2-2腔体阀关条件
OUT 602.11  ; #2-2腔体阀开[A]
LD TR0
LD D1096.06  ; #2腔体机构关电池抽气阀（自动步）
AND H31.01  ; #2-2电池泄漏
LD D1096.07  ; #2腔体机构开电池注氦阀（自动步）
AND H31.03  ; #2-2电池注氦超时
ORLD
OR D1100.03  ; #2腔体机构关闭#2-2腔体阀（自动单检步）
LD D1104.04  ; #2腔体机构正压开腔体阀/负压关腔体阀/氦检阀打开
LD D1097.01  ; #2腔体机构清氦需求判定（自动步）
OR P_On
AND H5.15  ; 腔体模式（0-正压 1-负压）
LD D1100.11  ; #2腔体机构关闭#2-1腔体阀/清氦判定（自动单检步）
ANDNOT P_On
ORLD
LDNOT D1100.11  ; #2腔体机构关闭#2-1腔体阀/清氦判定（自动单检步）
AND D1101.07  ; #2腔体机构清氦需求判定（自动单检步）
ANDNOT D1097.01  ; #2腔体机构清氦需求判定（自动步）
ANDNOT P_On
ORLD
ANDLD
ORLD
LD D1096.05  ; #2腔体机构腔体抽气阀打开/延时开电池抽气阀（自动步）  // #1-2无料时不测试
ANDNOT H30.01  ; #2-2腔体有料记忆
ORLD
ANDLD
OUT 512.11  ; #2-2腔体阀关条件
LD TR0
LD 512.11  ; #2-2腔体阀关条件
OR 612.11  ; #2-2腔体阀关[A]
ANDLD
ANDNOT 821.13  ; #2-2腔体阀关到位标志
ANDNOT 502.11  ; #2-2腔体阀开条件
OUT 612.11  ; #2-2腔体阀关[A]

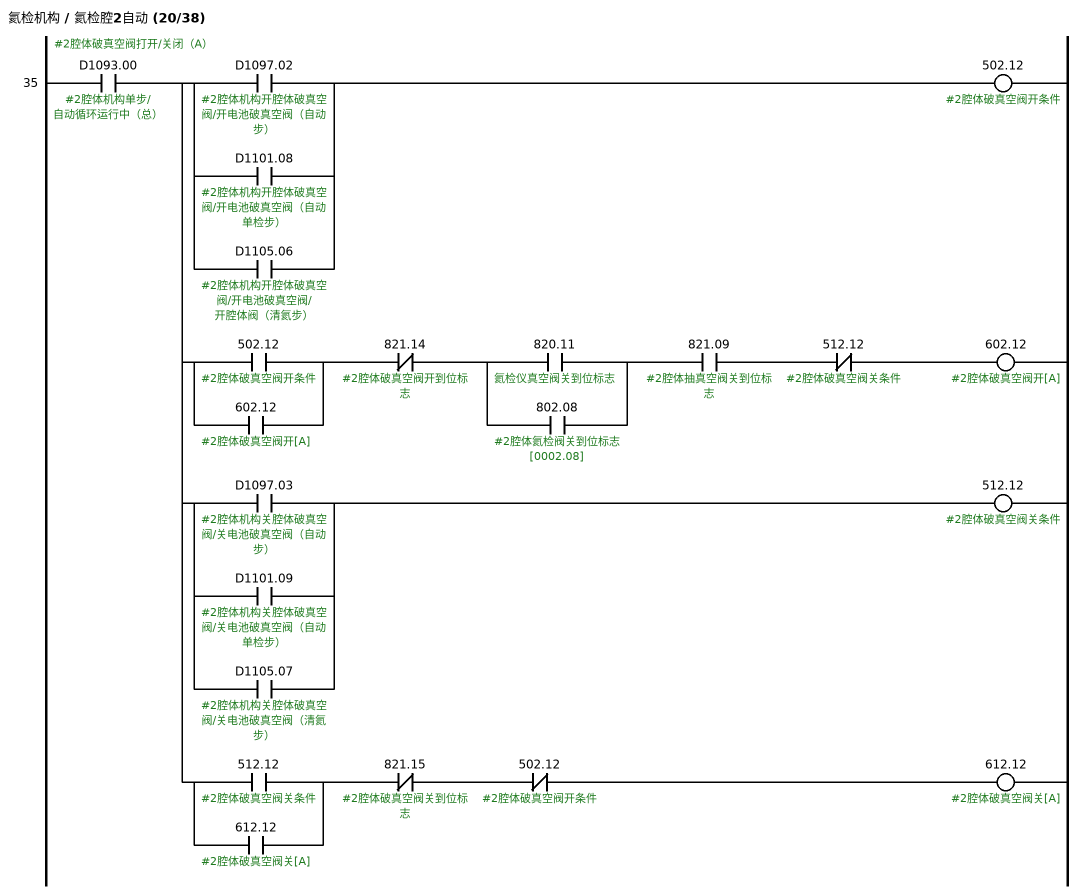
; rung 35: #2腔体破真空阀打开/关闭（A）
LD D1093.00  ; #2腔体机构单步/自动循环运行中（总）
OUT TR0
LD D1097.02  ; #2腔体机构开腔体破真空阀/开电池破真空阀（自动步）
OR D1101.08  ; #2腔体机构开腔体破真空阀/开电池破真空阀（自动单检步）
OR D1105.06  ; #2腔体机构开腔体破真空阀/开电池破真空阀/开腔体阀（清氦步）
ANDLD
OUT 502.12  ; #2腔体破真空阀开条件
LD TR0
LD 502.12  ; #2腔体破真空阀开条件
OR 602.12  ; #2腔体破真空阀开[A]
ANDLD
ANDNOT 821.14  ; #2腔体破真空阀开到位标志
LD 820.11  ; 氦检仪真空阀关到位标志
OR 802.08  ; #2腔体氦检阀关到位标志[0002.08]
ANDLD
AND 821.09  ; #2腔体抽真空阀关到位标志
ANDNOT 512.12  ; #2腔体破真空阀关条件
OUT 602.12  ; #2腔体破真空阀开[A]
LD TR0
LD D1097.03  ; #2腔体机构关腔体破真空阀/关电池破真空阀（自动步）
OR D1101.09  ; #2腔体机构关腔体破真空阀/关电池破真空阀（自动单检步）
OR D1105.07  ; #2腔体机构关腔体破真空阀/关电池破真空阀（清氦步）
ANDLD
OUT 512.12  ; #2腔体破真空阀关条件
LD TR0
LD 512.12  ; #2腔体破真空阀关条件
OR 612.12  ; #2腔体破真空阀关[A]
ANDLD
ANDNOT 821.15  ; #2腔体破真空阀关到位标志
ANDNOT 502.12  ; #2腔体破真空阀开条件
OUT 612.12  ; #2腔体破真空阀关[A]

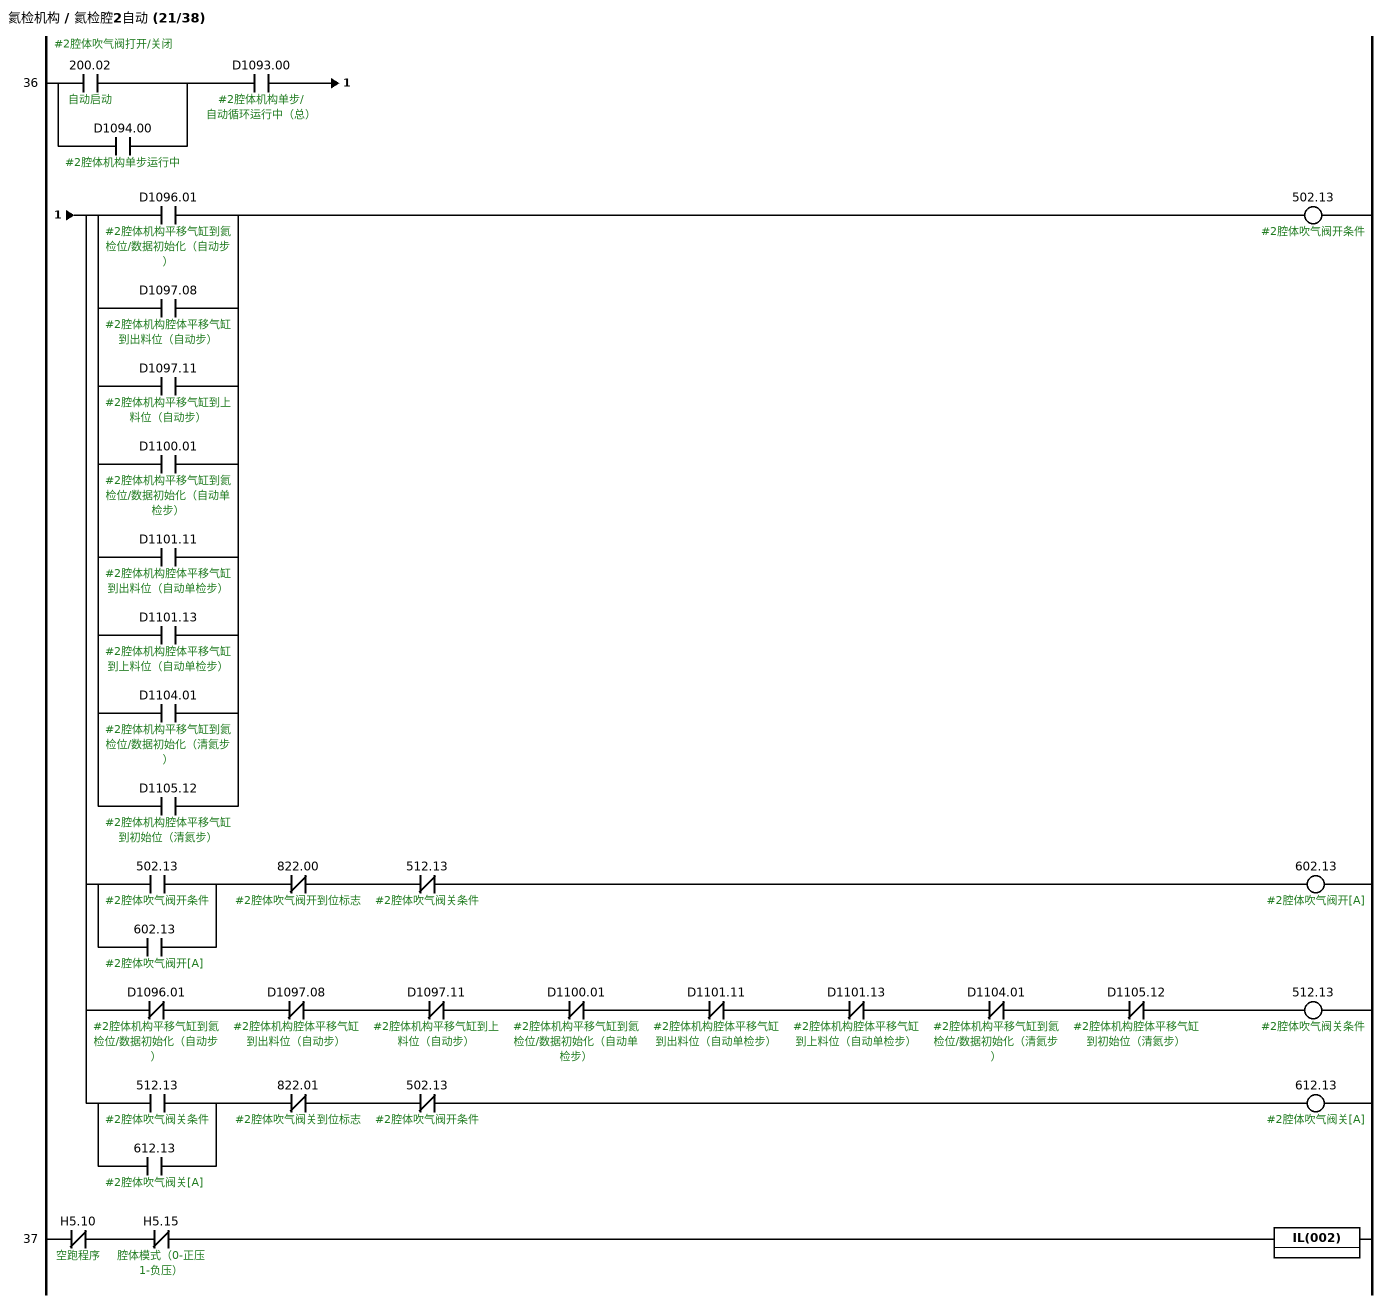
; rung 36: #2腔体吹气阀打开/关闭
LD 200.02  ; 自动启动
OR D1094.00  ; #2腔体机构单步运行中
AND D1093.00  ; #2腔体机构单步/自动循环运行中（总）
OUT TR0
LD D1096.01  ; #2腔体机构平移气缸到氦检位/数据初始化（自动步）
OR D1097.08  ; #2腔体机构腔体平移气缸到出料位（自动步）
OR D1097.11  ; #2腔体机构平移气缸到上料位（自动步）
OR D1100.01  ; #2腔体机构平移气缸到氦检位/数据初始化（自动单检步）
OR D1101.11  ; #2腔体机构腔体平移气缸到出料位（自动单检步）
OR D1101.13  ; #2腔体机构腔体平移气缸到上料位（自动单检步）
OR D1104.01  ; #2腔体机构平移气缸到氦检位/数据初始化（清氦步）
OR D1105.12  ; #2腔体机构腔体平移气缸到初始位（清氦步）
ANDLD
OUT 502.13  ; #2腔体吹气阀开条件
LD TR0
LD 502.13  ; #2腔体吹气阀开条件
OR 602.13  ; #2腔体吹气阀开[A]
ANDLD
ANDNOT 822.00  ; #2腔体吹气阀开到位标志
ANDNOT 512.13  ; #2腔体吹气阀关条件
OUT 602.13  ; #2腔体吹气阀开[A]
LD TR0
ANDNOT D1096.01  ; #2腔体机构平移气缸到氦检位/数据初始化（自动步）
ANDNOT D1097.08  ; #2腔体机构腔体平移气缸到出料位（自动步）
ANDNOT D1097.11  ; #2腔体机构平移气缸到上料位（自动步）
ANDNOT D1100.01  ; #2腔体机构平移气缸到氦检位/数据初始化（自动单检步）
ANDNOT D1101.11  ; #2腔体机构腔体平移气缸到出料位（自动单检步）
ANDNOT D1101.13  ; #2腔体机构腔体平移气缸到上料位（自动单检步）
ANDNOT D1104.01  ; #2腔体机构平移气缸到氦检位/数据初始化（清氦步）
ANDNOT D1105.12  ; #2腔体机构腔体平移气缸到初始位（清氦步）
OUT 512.13  ; #2腔体吹气阀关条件
LD TR0
LD 512.13  ; #2腔体吹气阀关条件
OR 612.13  ; #2腔体吹气阀关[A]
ANDLD
ANDNOT 822.01  ; #2腔体吹气阀关到位标志
ANDNOT 502.13  ; #2腔体吹气阀开条件
OUT 612.13  ; #2腔体吹气阀关[A]
; rung 37
LDNOT H5.10  ; 空跑程序
ANDNOT H5.15  ; 腔体模式（0-正压 1-负压）
IL(002)

